(* Logix 5000 project; controller STAT 1756-L72 rev 20.12; software revision 20.04; part 23 of 34 *)
(* tags used below, declared in another part *)
   av320 : BOOL;
   BITMW2 : BOOL;
   DateTime : DINT[7];   // DINT array tag for retrieve wallclock time through GSV created during conversion
   ForceStatus : INT;   // INT tag to retrieve Force enabled value through GSV created during conversion
   FRANCK : BOOL;
   lastmonth_put1 : DINT;
   lastmonth_put2 : DINT;
   lastmonth_totosmose : DINT;
   lastmonth_totq1 : DINT;
   lastmonth_totq2 : DINT;
   lastmonth_totq3 : DINT;
   mem_vent_yesterdsay : REAL;
   memjour : DINT;
   ONS1 : DINT;
   op010 : DINT;
   passage_jourmois : BOOL;
   PM3 : BOOL;
   PM4 : BOOL;
   real : REAL;
   S_AV320_V1_FC_C : BOOL;
   S_AV320_V1_FC_O : BOOL;
   S_AV320_V2_FC_C : BOOL;
   S_AV320_V2_FC_O : BOOL;
   s_flow_lancy_L1 : REAL;
   s_flow_lancy_L2 : REAL;
   s_flow_lancy_L3 : REAL;
   s_lvl_op006 : REAL;
   s_lvl_op007 : REAL;
   s_lvl_op008 : REAL;
   s_lvl_op009 : REAL;
   s_lvl_op010 : REAL;
   s_lvl_op011 : REAL;
   s_lvl_pellets_L4 : REAL;
   s_tot_vent_day : REAL;
   scp_flow_lancy_L1 : SCP;
   scp_flow_lancy_L2 : SCP;
   scp_flow_lancy_L3 : SCP;
   scp_flvl_op006 : SCP;
   scp_flvl_op007 : SCP;
   scp_flvl_op008 : SCP;
   scp_flvl_op009 : SCP;
   scp_flvl_op010 : SCP;
   scp_flvl_op011 : SCP;
   scp_lvl_pellets_L4 : SCP;
   stat_L1 : DINT[20];
   STAT_L2 : DINT[20];
   STAT_L3 : DINT[20];
   Status : INT;   // INT tag to retrieve Status value through GSV created during conversion
   tot_pulse_venturi : REAL;
(* ibt, continued *)

ROUTINE StatusFile   (* ladder *)
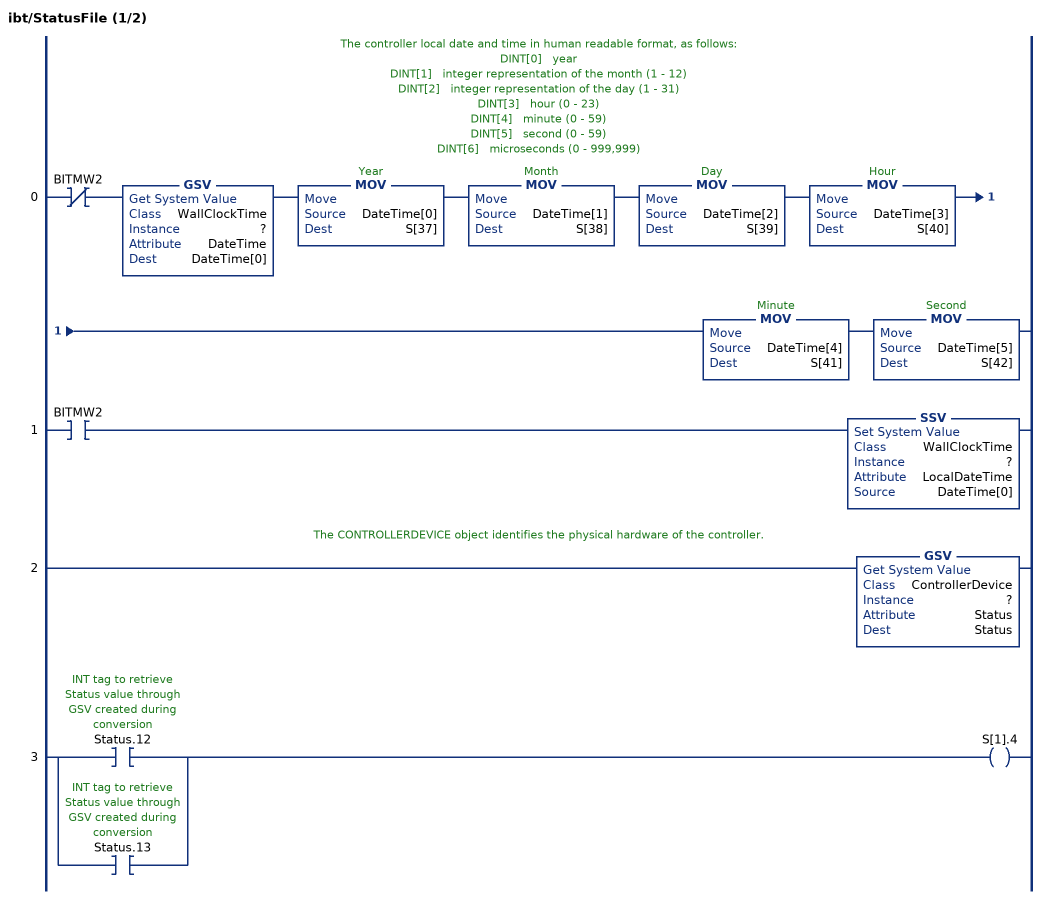
   // The controller local date and time in human readable format, as follows:
   // DINT[0] 	year
   // DINT[1] 	integer representation of the month (1 - 12)
   // DINT[2] 	integer representation of the day (1 - 31)
   // DINT[3] 	hour (0 - 23)
   // DINT[4] 	minute (0 - 59)
   // DINT[5] 	second (0 - 59)
   // DINT[6] 	microseconds (0 - 999,999)
   0: XIO(BITMW2)GSV(WallClockTime,?,DateTime,DateTime[0])MOV(DateTime[0],S[37])MOV(DateTime[1],S[38])MOV(DateTime[2],S[39])MOV(DateTime[3],S[40])MOV(DateTime[4],S[41])MOV(DateTime[5],S[42]);
   1: XIC(BITMW2)SSV(WallClockTime,?,LocalDateTime,DateTime[0]);
   // The CONTROLLERDEVICE object identifies the physical hardware of the controller.
   2: GSV(ControllerDevice,?,Status,Status);
   3: [XIC(Status.12) ,XIC(Status.13) ]OTE(S[1].4);
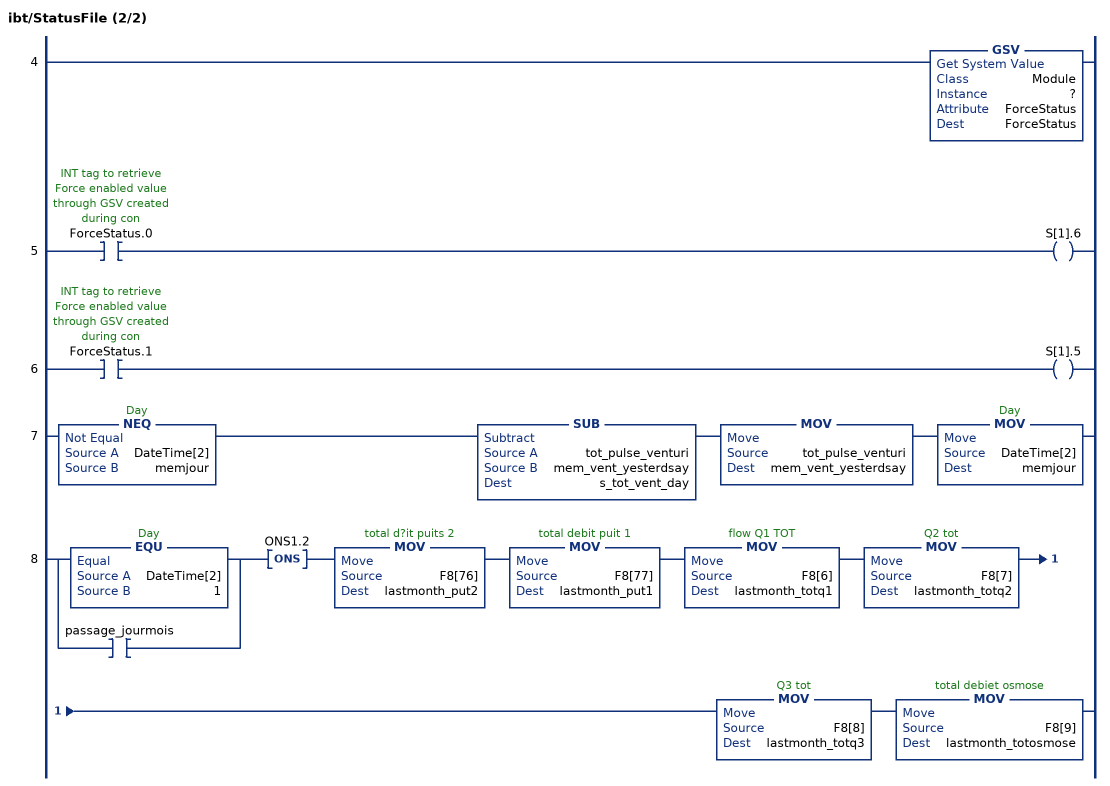
   4: GSV(Module,?,ForceStatus,ForceStatus);
   5: XIC(ForceStatus.0)OTE(S[1].6);
   6: XIC(ForceStatus.1)OTE(S[1].5);
   7: NEQ(DateTime[2],memjour)SUB(tot_pulse_venturi,mem_vent_yesterdsay,s_tot_vent_day)MOV(tot_pulse_venturi,mem_vent_yesterdsay)MOV(DateTime[2],memjour);
   8: [EQU(DateTime[2],1) ,XIC(passage_jourmois) ]ONS(ONS1.2)MOV(F8[76],lastmonth_put2)MOV(F8[77],lastmonth_put1)MOV(F8[6],lastmonth_totq1)MOV(F8[7],lastmonth_totq2)MOV(F8[8],lastmonth_totq3)MOV(F8[9],lastmonth_totosmose);
END_ROUTINE
END_PROGRAM

PROGRAM LANCY   (* main routine Lancy *)
VAR
   B3 : DINT[35] := ([1] := 2#0000_0000_0000_0000_0000_0010_0110_1001, [2] := 2#0000_0000_0000_0000_0000_0000_0000_0010, [3] := 2#0000_0000_0000_0000_0010_0001_1000_1000, [5] := 2#0000_0000_0000_0000_0000_0000_0000_0111, [6] := 2#0000_0000_0000_0000_0000_0100_0111_1110, [8] := 2#0000_0000_0000_0000_0000_0000_0000_1110, [10] := 2#0000_0000_0000_0000_1000_0000_0000_0000, [11] := 2#0000_0000_0000_0000_0000_0000_0000_1000, [25] := 2#0000_0000_0000_0000_0011_0000_0011_0000, [29] := 2#0000_0000_0000_0000_0010_0001_0000_0000, [31] := 2#0000_0000_0000_0000_0000_0100_0001_0000, [33] := 2#0000_0000_0000_0000_0000_0000_0001_1100, [34] := 2#0000_0000_0000_0000_0000_0010_0000_0000);
        [0].0   // res
        [0].1   // remplace L106E reactor tank T100 LE 106 E low level alarm
        [0].2   // remplace reactor tank T100 LE106 D
        [0].3   // remplace reactor tank T100 LE106 C
        [0].4   // remplace reactor tank T100 LE106 B
        [0].5   // remplace reactor tank T100 LE106 A
        [0].15   // ARRET POUR ENTRETIEN
        [2].0   // marche pmp puisard L123 sur debit venturi
        [2].1   // marche pmp puisard L123 sur niveau
        [2].3   // lvl orange atteint
        [2].4   // presence 1 niveau orange
        [2].5   // lvl rouge atteint
        [2].6   // changement dans les niveaux orange et rouge
        [2].7   // changement orange
        [2].8   // changement 1 niveau rouge
        [3].0   // L1 level point LE337 A
        [3].1   // L1 level point LE337 B
        [3].2   // L1 level point LE337 C
        [3].3   // L1 level point LE337 D
        [3].4   // L1 level point LE337 E
        [3].5   // L2 level point LE327 A
        [3].6   // L2 level point LE327 B
        [3].7   // L2 level point LE327 C
        [3].8   // L2 level point LE327 D
        [3].9   // L2 level point LE327 E
        [3].10   // L3 level point LE317 A
        [3].11   // L3 level point LE317 B
        [3].12   // L3 level point LE317 C
        [3].13   // L3 level point LE317 D
        [3].14   // L3 level point LE317 E
        [4].0   // L4 level point LE 400 A
        [4].1   // L4 level point LE 400 B
        [4].2   // L4 level point LE 400 C
        [4].3   // L4 level point LE 400 D
        [4].4   // L4 level point LE 400 E
        [5].0   // L4 Filtrate return Valve LV 410
        [5].1   // LV 410 open
        [5].2   // LV 410 closed
        [6].0   // op008->ph bak no default
        [6].1   // op008->holding tank no default
        [6].2   // op008->reactor no default
        [6].3   // ok L1 -> OP008
        [6].4   // ok L2 -> OP008
        [6].5   // ok L3 -> OP008
        [6].6   // ok L1->holding tank eau rinçage
        [6].7   // op008 -> L1 ok
        [6].9   // OP008 -> L3 OK
        [7].0   // pmp OP008 ok for run
        [7].3   // rinçage tuyauterie HT
        [8].0   // filtrate lift station T160 LE165 A
        [8].1   // filtrate lift station T160 LE165 B
        [8].2   // filtrate lift station T160 LE165 C
        [8].3   // filtrate lift station T160 LE165 D
        [9].0   // BP L1 -> holding tank
        [9].1   // de supervis BP L1-> OP008
        [9].2   // de superv BP L2 -> OP008
        [9].3   // de superv BP L3 -> OP008
        [9].4   // de superv BP OP008 -> reactor
        [9].6   // start].stop
        [10].11   // demande stop soude
        [10].12   // apport soude demande de marche
        [10].13   // marche soude ouverture vanne
        [10].14   // ons
        [10].15   // ons
        [25].0   // reactor tank T100 high level alarm
        [25].1   // reactor tank T100 high level alarm horn silence
        [25].2   // reactor tank T100 low level alarm
        [25].3   // reactor tank T100 low level alarm horn silence
        [25].4   // holding tank T130 low level alarm
        [25].5   // holding tank T130 low level alarm horn silence
        [25].6   // clear filtrate receiver tank T260 high level alarm
        [25].7   // clear filtrate receiver tank T260 high level alarm horn simence
        [25].10   // cloudy filtrate receiver tank T270 high level alarm
        [25].11   // cloudy filtrate receiver tank T270 high level alarm horn silence
        [25].12   // vacuum pup suction line high level alarm
        [25].13   // vacuum pup suction line high level alarm horn silence
        [25].14   // filtrate lift station high level alarm
        [25].15   // filtrate lift station high level alarm horn silence
        [26].0   // L3 high level alarm
        [26].1   // L3 high level alarm horn silence
        [26].4   // L3 low level alarm
        [26].5   // L3 low level alarm horn silence
        [26].6   // L2 high level alarm
        [26].7   // L2 high level alarm horn silence
        [26].8   // L2 low level alarm
        [26].9   // L2 low level alarm horn silence
        [26].10   // L1 high level alarm
        [26].11   // L1 high level alarm horn silence
        [26].14   // L1 low level alarm
        [26].15   // L1 low level alarm horn silence
        [27].0   // surge tank T150 turbidity control alarm
        [27].1   // surge tank T150 turbidity control alarm horn silence
        [27].2   // Mixer M110 failure alarm
        [27].3   // Mixer M110 failure alarm horn silence
        [27].4   // M120 overcurrent alarm
        [27].5   // M120 overcurrent alarm silence horn
        [27].8   // P170 overcurrent alarm
        [27].9   // P170 overcurrent alarm horn silence
        [27].10   // P180 overcurrent alarm
        [27].11   // P180 overcurrent alarm horn silence
        [27].12   // P210 overcurrent alarm
        [27].13   // P210 overcurrent alarm horn silence
        [27].14   // P220 overcurrent alarm
        [27].15   // P220 overcurrent alarm horn silence
        [28].2   // P230 overcurrent alarm
        [28].3   // P230 overcurrent alarm horn silence
        [28].4   // P240 overcurrent alarm
        [28].5   // P240 overcurrent alarm horn silence
        [28].6   // F200 overcurrent alarm
        [28].7   // F200 overcurrent alarm horn silence
        [28].8   // P250 overcurrent alarm
        [28].9   // P250 overcurrent alarm horn silence
        [28].13   // clear filtrate pumps P210 & P220 failure alarm horn silence
        [28].15   // cloudy flitrate pump P230 & P240 failure alarm horn silence
        [29].0   // filtrate lift pump P170 failure alarm
        [29].1   // filtrate lift pump P170 failure alarm horn silence
        [29].6   // 0cr
        [29].8   // 2cr
        [29].9   // 3 cr
        [29].10   // 4 cr
        [29].12   // 6 cr
        [29].13   // 7 cr
        [30].1   // 9 cr
        [30].2   // 10 CR
        [30].6   // reactor tank T100 Level B].C diffential disable relay
        [30].7   // vacuum pump P250 seal water low flow alarm
        [30].10   // vacuum pump P250 seal water low flow alarm horn silenc
        [30].11   // horn auxiliaire 1
        [30].12   // horn auxiliaire 2
        [30].13   // horn auxiliaire 3
        [30].14   // horn auxiliaire 4
        [30].15   // horn auxiliaire 5
        [31].4   // clignotant
        [31].6   // delay off timer filtrate lift pump seal water valve
        [31].7   // delay off timer filtrate lift pump P170 failure alarm
        [31].8   // tempo clear filtrate pumps seal water off delay
        [31].9   // cloudy flitrate pumps delay off timer
        [31].10   // vacuum pump P250 delay on
        [31].11   // vacuum pump seal water valve SV255 delay off timer
        [31].15   // clear filtrate pumps P210 failure alarm
        [32].0   // clear filtrate pumps P220 failure alarm
        [32].1   // tempo clear filtrate pumps P210 failure alarm delay
        [32].2   // tempo clear filtrate pumps P220 failure alarm delay
        [32].3   // cloudy flitrate pump P230 failure alarm
        [32].4   // cloudy flitrate pump P240 failure alarm
        [32].5   // cloudy flitrate pump P230 failure alarm delay
        [32].8   // cloudy flitrate pump P240 failure alarm delay
        [32].11   // vacuum pump P250 low flow delay timer
        [32].12   // shearing mixer M120 off delay timer
        [32].13   // M110 not running
        [32].14   // Mixer M110 failure delay
        [33].2   // L1 active
        [33].3   // L2 active
        [33].4   // L3 active
        [33].5   // L1 active & >level B
        [33].6   // L2 active & >level B
        [33].7   // L3 active & >level B
        [33].8   // All line not active
        [33].12   // AV valve override
        [33].13   // system high relay
        [33].14   // system high silence
        [33].15   // system high high level alarm
        [34].0   // system high high level alarm silence
        [34].1   // regenerate caustic available alarm at holding tank T130
        [34].2   // regenerate caustic available at holding tank T130 alarm silence
        [34].6   // L4 active
        [34].7   // L4 active & >level B
        [34].8   // 11 cr
        [34].9   // 12 cr
        [34].10   // L4 high level alarm
        [34].11   // L4 high level alarm horn silence
        [34].12   // L4 low level alarm
        [34].13   // L4 low level alarm horn silence
        [10].9   // demande soude station
   C5 : COUNTER[10];
        [0].DN   // g
        [0].PRE   // y
   F8 : REAL[100] := ([1] := 324.85922, [2] := 2.0, [3] := 162.42961, [4] := -2.7111664, [5] := 105.0, [10] := 199.0041, [11] := 284.0703, [12] := 333.46686, [13] := 763.174, [14] := 438.31393, [15] := 310.28265);
        [0]   // jg
        [2]   // ratio venturi].filtrat
        [3]   // debit filtrat souhaité en 0.1m³].h
        [4]   // erreur debit filtrat 0.1 m³].h
        [5]   // consigne ouverture servo vanne filtrat
        [10]   // niveau op006
        [11]   // aux niveau op007
        [12]   // aux niveau op008
        [13]   // aux niveau op009
        [14]   // aux niveau op010
        [15]   // aux niveau op011
   N20 : DINT[50] := ([0] := -16384, [1] := 4, [5] := 2, [10] := 199, [11] := 284, [12] := 333, [13] := 762, [14] := 438, [15] := 309, [17] := 632, [20] := 7935, [22] := 388, [23] := 264, [25] := 4, [30] := 5, [32] := 199, [33] := 284, [34] := 333, [35] := 199, [37] := 284, [39] := 332, [40] := -1, [41] := 766, [42] := 3, [43] := 438, [45] := 311, [46] := 1, [47] := 763, [48] := 438, [49] := 310);
        [0]   // bit pour superv
        [1]   // DEFAUT PRIORITE 1
        [2]   // defaut niveau 2
        [5].0   // DEFAULT
        [5].1   // NEW DEFAULT
        [9].1   // ack STOCK
        [10]   // niveau op006
        [11]   // niveau op007
        [12]   // niveau op008
        [13]   // niveau op009
        [14]   // niveau op010
        [15]   // niveau op011
        [16].1   // level holding tank
        [16].2   // valve positie
        [20].0   // reactor tank T100 high level alarm
        [20].1   // reactor tank T100 low level alarm
        [20].2   // holding tank T130 low level alarm
        [20].3   // clear filtrate receiver tank T260 high level alarm
        [20].4   // cloudy filtrate receiver tank T270 high level alarm
        [20].5   // vacuum pup suction line high level alarm
        [20].6   // filtrate lift station high level alarm
        [20].7   // L3 high level alarm
        [20].8   // L3 low level alarm
        [20].9   // L2 high level alarm
        [20].10   // L2 low level alarm
        [20].11   // L1 high level alarm
        [20].12   // L1 low level alarm
        [20].13   // surge tank T150 turbidity control alarm
        [20].14   // Mixer M110 failure alarm
        [20].15   // M120 overcurrent alarm
        [21].0   // P170 overcurrent alarm
        [21].1   // P180 overcurrent alarm
        [21].2   // P210 overcurrent alarm
        [21].3   // P220 overcurrent alarm
        [21].4   // P230 overcurrent alarm
        [21].5   // P240 overcurrent alarm
        [21].6   // F200 overcurrent alarm
        [21].7   // P250 overcurrent alarm
        [21].8   // filtrate lift pump P170 failure alarm
        [21].9   // vacuum pump P250 seal water low flow alarm
        [21].10   // L4 high level alarm
        [21].11   // L4 low level alarm
        [21].12   // clear filtrate pumps P210 failure alarm
        [21].13   // clear filtrate pumps P220 failure alarm
        [21].14   // cloudy flitrate pump P230 failure alarm
        [21].15   // cloudy flitrate pump P240 failure alarm
        [22].0   // system high relay
        [22].1   // system high high level alarm
        [22].2   // regenerate caustic available alarm at holding tank T130
        [22].3   // DEF POS VANNE SILO
        [22].4   // DEF POS VANNE BOUILLOIRE
        [22].5   // DEF POSIT ST VA1
        [22].6   // DEF POSIT ST VA 2
        [22].7   // DEF POSIT ST VA3
        [22].8   // DEF POSIT ST VA4
        [22].9   // DEF POSIT ST VA5
        [22].10   // DEF POSIT ST VA6
        [22].11   // DEF POSIT ST VA7
        [22].14   // DEF PP1 STAT
        [23].12   // mixer arreté pour Franck mixer stil pour herman
        [25].0   // reactor tank T100 high level alarm
        [25].1   // reactor tank T100 low level alarm
        [25].2   // holding tank T130 low level alarm
        [25].3   // clear filtrate receiver tank T260 high level alarm
        [25].4   // cloudy filtrate receiver tank T270 high level alarm
        [25].5   // vacuum pup suction line high level alarm
        [25].6   // filtrate lift station high level alarm
        [25].7   // L3 high level alarm
        [25].8   // L3 low level alarm
        [25].9   // L2 high level alarm
        [25].10   // L2 low level alarm
        [25].11   // L1 high level alarm
        [25].12   // L1 low level alarm
        [25].13   // surge tank T150 turbidity control alarm
        [25].14   // Mixer M110 failure alarm
        [25].15   // M120 overcurrent alarm
        [26].0   // P170 overcurrent alarm
        [26].1   // P180 overcurrent alarm
        [26].2   // P210 overcurrent alarm
        [26].3   // P220 overcurrent alarm
        [26].4   // P230 overcurrent alarm
        [26].5   // P240 overcurrent alarm
        [26].6   // F200 overcurrent alarm
        [26].7   // P250 overcurrent alarm
        [26].8   // filtrate lift pump P170 failure alarm
        [26].9   // vacuum pump P250 seal water low flow alarm
        [26].10   // L4 high level alarm
        [26].11   // L4 low level alarm
        [26].12   // clear filtrate pumps P210 failure alarm
        [26].13   // clear filtrate pumps P220 failure alarm
        [26].14   // cloudy flitrate pump P230 failure alarm
        [26].15   // cloudy flitrate pump P240 failure alarm
        [27].0   // system high relay
        [27].1   // system high high level alarm
        [27].2   // regenerate caustic available alarm at holding tank T130
        [27].3   // DEF POS VANNE SILO
        [27].4   // DEF POS VANNE BOUILLOIRE
        [27].5   // DEF POSIT ST VA1
        [27].6   // DEF POSIT ST VA 2
        [27].7   // DEF POSIT ST VA3
        [27].8   // DEF POSIT ST VA 4
        [27].9   // DEF POSIT ST VA5
        [27].10   // DEF POSIT ST VA6
        [27].11   // DEF POSIT ST VA7
        [27].14   // DEF PP1 STAT
        [30]   // NOMBRE DE DEFAUTS
        [31]   // MEMO NOMBRE DE DEFAUTS
        [32]   // op006
        [33]   // op007
        [34]   // op008
        [36]   // delta viveau op006
        [38]   // delta viveau op007
        [40]   // delta viveau op008
        [42]   // delta viveau op009
        [44]   // delta niveau op010
        [46]   // delta niveau op011
        [47]   // op009
        [48]   // op010
        [49]   // op011
   N7 : DINT[150] := ([1] := -250, [2] := 994, [3] := 958, [4] := -250, [5] := 982, [6] := 994, [7] := 958, [8] := 982, [10] := 165, [11] := -25, [12] := 888, [13] := 609, [15] := 955, [16] := -250, [17] := -250, [18] := 632, [19] := 269, [20] := 105, [21] := -16384, [23] := 894, [26] := 16, [29] := 525, [30] := 600, [31] := 400, [32] := 575, [33] := 350, [34] := 609, [35] := 30, [36] := 49, [37] := 65, [39] := 2, [40] := 1170, [45] := 754, [50] := 14, [57] := 10, [60] := 438, [61] := 6, [62] := 173, [64] := 20, [65] := 2048, [70] := 7, [71] := 27, [72] := 10, [73] := 11, [74] := 137, [75] := 100, [78] := 5, [90] := 6, [91] := 609, [94] := 5, [96] := 45, [98] := 45, [99] := 45, [101] := 5, [102] := 5, [103] := 5, [104] := 5, [105] := 5, [106] := 5, [110] := 8192,
        [111] := 32, [112] := 1, [113] := 7, [114] := 137, [115] := 250, [118] := 5, [140] := 21, [141] := 780, [142] := 800);
        [12]   // niveau reacteur Lancy E 905 / changer le D920 /12/07/16 C965 B975 A985
        [0]   // mojilhk
        [10]   // debit filtrat filtre-presse 0.1 m³].h
        [11]   // position servo vanne filtrat
        [13]   // niveau puisard L123
        [16]   // hac turbidity 0-1000 mtu
        [17]   // optek turbidity 0-1000 mtu
        [18]   // niveau BUFFER VOOR FILTER PERS
        [19]   // LEVEL FLITRAAT WATER FROM FILTERPERS
        [20]   // cmd position vanne filtrat
        [21]   // memo
        [25]   // vers stock quantité soude demandée
        [26].0   // vers plc stock demande de soude L1
        [26].1   // vers plc stock demande d'arret apport soude
        [26].2   // vers plc stock fc vanne apport soude décapage
        [26].3   // vers plc stock apport soude finit
        [26].4   // vers plc stock fc vanne apport soude décapage
        [29]   // niveau lift tank
        [36]   // memo debit venturi
        [38]   // diferrence debit venturi
        [45]   // soude restante
        [46].3   // de plc stock ouverture vanne soude
        [46].4   // de plc stock apport soude finit
        [46].5   // de plc stock apport soude occupé
        [46].6   // de plc stock apport soude accordé
        [46].7   // de plc stock soude vers l1
        [46].8   // de plc stock soude vers L2
        [46].9   // de plc stock soude vers L3
        [46].10   // de plc stock soude vers L4
        [46].11   // de plc stock soude vers STAT
        [50]   // debit venturi m³].h de IBT
        [51]   // reserver de IBT
        [52]   // reserver de IBT
        [53]   // reserver de IBT
        [54]   // reserver de IBT
        [55]   // reserver de IBT
        [60]   // vers ecotech op010
        [70]   // message ecriture IBT
        [90].0   // Mixer M110 failure alarm
        [90].1   // vers slc ibt marche pmp 1 puisard L123
        [90].2   // vers slc ibt marche pmp 2 puisard L123
        [90].3   // vers slc ibt stop pm3 et pm4
        [91]   // level puisard L1 2 3
        [94]   // pas à pas sequence ?? NAOH
        [95]   // DEBIT L1
        [96]   // DEBIT L2
        [97]   // DEBIT L3
        [98]   // TOTAL L 1 2 3
        [99]   // aux TOTAL L 1 2 3
        [100]   // pas à pas op008-> L4
        [101]   // pas a pas op008 -> Holding Tank
        [102]   // pas a pas op008 -> reactor
        [103]   // pas a pas L1 -> OP008
        [104]   // pas a pas L2 -> OP008
        [105]   // pas a pas L3 -> OP008
        [106]   // pas a pas renvoi eau nettoyage
        [107]   // op008 -> L1
        [108]   // op008 -> L2
        [109]   // op 008 L3
        [110]   // stock
        [131]   // MEMO AUX FLOW L1
        [132]   // MEMO AUX FLOW L2
        [133]   // MEMO AUX FLOW L2
        [134]   // MEMO AUX FLOW L3
        [135]   // MEMO AUX FLOW L3
        [140].0   // envoi defaut niv 1 present
        [140].1   // defaut niveau 2 present
        [140].2   // defaut rappel envoi
        [141]   // level high buffer fl
        [142]   // level high high buff
   N9 : DINT[200] := ([0] := 10, [1] := -1, [10] := 509, [11] := -32474, [14] := 1, [20] := 346, [21] := 1062, [23] := 4, [24] := -12, [30] := 484, [31] := 430, [33] := 4, [34] := -1, [36] := 10, [43] := 91, [60] := 2, [71] := 2349, [73] := 165, [74] := 93, [75] := -25, [76] := 609, [77] := -250, [78] := 49, [79] := 484, [80] := 199, [81] := 284, [82] := 333, [83] := 763, [84] := 438, [85] := 310, [86] := -16384, [87] := 35415, [88] := 43684, [89] := 888, [91] := 45, [94] := 930, [96] := -32346, [97] := 8614, [98] := 430, [99] := 3074, [100] := 4620, [101] := 61, [104] := 10, [107] := 270, [111] := 1, [112] := 1, [120] := 1, [121] := 1, [122] := -1, [134] := 3, [142] := 1, [143] := 9, [144] := 137, [145] := 4, [147] := 512, [148] := 5, [155] := 2, [160] := 7, [161] := 16, [162] := 1,
        [163] := 9, [164] := 137, [165] := 4, [168] := 5, [175] := 2, [180] := 7, [181] := 24, [182] := 1, [183] := 9, [184] := 137, [185] := 4, [188] := 5, [195] := 2);
        [21].0   // L2VA1 open
        [97].0   // L2VA1 open
        [100].16   // de superv Stop trajet L1 vers holding tank
        [21].1   // l2VA1 close
        [97].1   // l2VA1 close
        [97].8   // pp2 run
        [0]   // h,j;
        [0].0   // DE PLC STOCK L1 VA 4 FC O
        [0].1   // DE PLC STOCK L1 VA 4 FC F
        [0].2   // DE PLC STOCK L2 VA 4 FC O
        [0].3   // DE PLC STOCK L2 VA 4 FC F
        [2]   // de stock
        [3]   // defaut 2 stock
        [10]   // niveau decapage L1
        [11].0   // VA1 open
        [11].1   // VA1 close
        [11].2   // VA2 open
        [11].3   // VA2 close
        [11].4   // VA3 open
        [11].5   // VA3 close
        [11].6   // reserve
        [11].7   // reserve
        [11].8   // pp1 run
        [11].9   // pp1 TH
        [11].10   // pp2 run
        [11].11   // pp2 TH
        [11].12   // soude passée
        [11].14   // marche renvoi eau rinçage bain decap ligne 1
        [11].15   // arret renvoi eau rinçage bain decap ligne 1
        [12]   // total soude passé vers op008
        [14]   // reserve de ligne 1
        [20]   // level decap ligne 2
        [21].2   // L2 VA2 open
        [21].3   // VA2 close
        [21].4   // VA3 open
        [21].5   // VA3 close
        [21].6   // VA4 open
        [21].7   // VA4 close
        [21].8   // pp1 run
        [21].9   // pp1 TH
        [21].10   // pp2 run
        [21].11   // pp2 TH
        [21].12   // soude passée
        [22]   // total soude passé vers op008
        [24]   // def niv 1 L2
        [25]   // def niv 2 L2
        [30]   // niveau decapage L3
        [31].0   // VA1 open
        [31].1   // VA1 close
        [31].2   // VA2 open
        [31].3   // VA2 close
        [31].4   // VA3 open
        [31].5   // VA3 close
        [31].6   // VA4 open
        [31].7   // VA4 close
        [31].8   // pp1 run
        [31].9   // pp1 TH
        [31].10   // pp2 run
        [31].11   // pp2 TH
        [31].12   // soude passée
        [32]   // total soude passé vers op008
        [33]   // quantité eau de ligne
        [34]   // defaut niv 1 L3
        [35]   // defaut niv 2 L3
        [42]   // quantité soude demandée
        [43]   // quantite soude passé
        [50].0   // open L1VA4
        [50].1   // open L2 VA4
        [60].0   // retour alarm niv 1 vu
        [60].1   // retour alarm niv 2 vu
        [60].2   // retour alarm niv 3 vu
        [70]   // consigne en % decap L4
        [70].0   // defaut niv 1
        [71]   // conversion m³ en % dec L4
        [80]   // niveau op006
        [81]   // niveau op007
        [82]   // niveau op008
        [83]   // niveau op009
        [84]   // niveau op010
        [85]   // niveau op011
        [86].0   // lvl rouge OP006
        [86].1   // lvl orange OP006
        [86].2   // lvl rouge OP007
        [86].3   // lvl orange OP007
        [86].4   // lvl rouge OP008
        [86].5   // lvl orange OP008
        [86].6   // lvl rouge OP009
        [86].7   // lvl orange OP009
        [86].8   // lvl rouge OP010
        [86].9   // lvl orange OP010
        [86].10   // lvl rouge OP011
        [86].11   // lvl orange OP011
        [86].12   // change display spervision
        [86].13   // level op008 too low
        [87].0   // vers supervision AV 147 open
        [87].1   // vers supervision AV 320 open
        [87].2   // vers supervision LV 325 open
        [87].3   // vers supervision AV 330 open
        [87].4   // vers supervision LV 335 open
        [87].5   // vers supervision AV 310 open
        [87].6   // vers supervision LV 315 open
        [87].7   // vers supervision clear filtrate P210
        [87].8   // vers supervision clear filtrate pumps P210 failure
        [87].9   // vers supervision clear filtrate P220
        [87].10   // vers supervision clear filtrate pumpsP220 failure
        [87].11   // vers supervision cloudy filtrate P230
        [87].12   // vers supervision cloudy flitrate pump P230 failure
        [87].13   // vers supervision cloudy filtrate P240
        [87].14   // vers supervision cloudy flitrate pump P240 failure
        [87].15   // vers supervision
        [88].0   // vers supervision filtrate lift pump P170
        [88].1   // vers supervision P170 overcurrent alarm
        [88].2   // vers supervision filtrate lift pump P180
        [88].3   // vers supervision P180 overcurrent alarm
        [88].4   // vers supervision ST VA1 open
        [88].5   // vers supervision ST VA1 close
        [88].6   // vers supervision ST VA2 open
        [88].7   // vers supervision ST VA2 close
        [88].8   // vers supervision ST VA3 open
        [88].9   // vers supervision ST VA3 close
        [88].10   // vers supervision ST VA4 open
        [88].11   // vers supervision ST VA4 close
        [88].12   // vers supervision ST VA5 open
        [88].13   // vers supervision ST VA5 close
        [88].14   // vers supervision ST VA6 open
        [88].15   // vers supervision ST VA6 close
        [89]   // vers supervission niveau reacteur Lancy
        [90]   // DEBIT L1
        [91]   // DEBIT L2
        [92]   // DEBIT L3
        [93]   // level holding tank
        [94]   // level Ph bak
        [95]   // total soude passé vers op008
        [96].0   // L1 VA1 open
        [96].1   // L1 VA1 closed
        [96].2   // L1 va2 ouverte
        [96].3   // L1 va2 closed
        [96].4   // L1 va3 ouverte
        [96].5   // L1 va3 closed
        [96].6   // L1 VA4 open
        [96].7   // L1 VA4 close
        [96].8   // L1 PP1 RUN
        [97].2   // L2 VA2 open
        [97].6   // L2 VA4 open
        [97].7   // L2 VA4 close
        [98].0   // L3 VA1 open
        [98].1   // L3 VA1 closed
        [98].2   // L3 VA2 open
        [98].4   // L3 VA3 open
        [98].6   // L3 VA4 open
        [98].7   // L3 VA4 closed
        [98].8   // L3 pp1 run
        [99].0   // vers supervision ST VA7 open
        [99].1   // vers supervision ST VA7 close
        [99].2   // vers suprt defaut protection pompe PP1
        [99].3   // vers suprt rotation pompe st PP1 op008
        [99].4   // op008 - > reactor en dmd ou en rinçage
        [99].5   // op008 - > reactor run
        [99].6   // op008 - > holding tank en dmd ou en rinçage
        [99].7   // op008 - > holding tank run
        [99].8   // op008 - > phbak en demande ou en rinçage
        [99].9   // op008 - > phbak run
        [99].10   // op008 - > reactor possible
        [99].11   // op008 - > holding tank possible
        [99].12   // op008 - > phbak possible
        [99].13   // de superv BP OP008 -> reactor
        [99].14   // de superv BP op008->holding T
        [99].15   // de superv bp op008->phbak
        [100].0   // vers superv level reactor too high
        [100].1   // vers superv level holding T too high
        [100].2   // vers superv level phbak too high
        [100].3   // open].close ST VA1
        [100].4   // BP L1 -> holding tank
        [100].6   // de supervis BP L1-> OP008
        [100].7   // de superv BP L2 -> OP008
        [100].8   // de superv BP L3 -> OP008
        [101]   // stock soude pellet L4
        [102]   // res flow naoh L2
        [103]   // res flow naoh L3
        [106]   // quantité naoh demander de L3
        [110]   // total soude passé vers op008
        [111].3   // de superv bp op008 ->L1
        [111].5   // de supervision BP op008 - > L3
        [113]   // res flow naoh L1
        [123]   // memo def 1 IBT
        [124]   // stock
        [125]   // lancy
        [140]   // ligne 1
        [155].0   // open L1 VA1
        [155].1   // open L1 VA2
        [155].2   // open L1 VA3
        [155].4   // DEFAULT FLOW NaOH FROM L1
        [155].5   // DEFAULT FLOW NaOH TO L1
        [160]   // ligne2
        [175].0   // open L2 VA1
        [175].1   // open L2 VA2
        [175].2   // open L2 VA3
        [175].4   // DEFAULT FLOW NaOH FROM L2
        [175].5   // DEFAULT FLOW NaOH TO L2
        [180]   // ligne 3
        [195].0   // open L3 VA1
        [195].1   // open L3 VA2
        [195].2   // open L3 VA3
        [195].3   // open L3 VA4
        [195].4   // DEFAULT FLOW NaOH FROM L3
        [195].5   // DEFAULT FLOW NaOH TO L3
        [195].6   // reactor tank T100 HH vers L3
   R6 : CONTROL[10];
   S : INT[164] := ([0] := 16#0004, [1] := 16#00e6, [2] := 16#9012, [3] := 16#a001, [4] := 16#4c06, [5] := 16#4000, [6] := 16#0021, [11] := 16#ffff, [12] := 16#ffff, [14] := 16#0046, [15] := 16#0b1e, [17] := 16#0002, [21] := 16#0002, [22] := 16#0003, [23] := 16#0001, [27] := 16#ffff, [28] := 16#ffff, [33] := 16#1808, [34] := 16#0002, [35] := 16#000b, [37] := 16#0775, [38] := 16#000c, [39] := 16#0018, [40] := 16#0006, [41] := 16#0021, [42] := 16#0008, [53] := 16#0006, [54] := 16#0021, [57] := 16#0191, [58] := 16#0002, [59] := 16#0006, [60] := 16#021d, [61] := 16#0002, [62] := 16#0007, [63] := 16#0401, [64] := 16#005f, [65] := 16#0010, [66] := 16#0200, [83] := 16#0046, [84] := 16#f000, [85] := 16#0001, [86] := 16#01a3);
   T4 : TIMER[100] := ([0].PRE := 9999, [0].ACC := 45, [1].PRE := 5000, [2].PRE := 10000, [3].PRE := 5000, [4].PRE := 5000, [5].PRE := 5000, [6].PRE := 5000, [7].PRE := 5000, [8].PRE := 5000, [9].PRE := 3000, [9].ACC := 3000, [9].EN := 1, [9].DN := 1, [10].PRE := 5000, [11].PRE := 3000, [12].PRE := 60000, [12].ACC := 50750, [12].EN := 1, [12].TT := 1, [13].PRE := 5000, [14].PRE := 2000, [14].ACC := 1500, [14].EN := 1, [14].TT := 1, [15].PRE := 10000, [15].ACC := 4000, [15].EN := 1, [15].TT := 1, [16].PRE := 60000, [16].ACC := 60000, [17].PRE := 450000, [18].PRE := 1200000, [18].ACC := 936100, [18].TT := 1, [18].DN := 1, [19].PRE := 30000, [19].ACC := 23850, [19].EN := 1, [19].TT := 1, [20].PRE := 700, [20].ACC := 600, [20].EN := 1, [20].TT := 1, [21].PRE := 5000, [22].PRE := 50000, [23].PRE := 50000, [24].PRE := 10000, [25].PRE := 5000, [26].PRE := 90000, [27].PRE := 3000, [27].ACC := 600, [27].EN := 1, [27].TT := 1, [28].PRE := 150000, [29].PRE := 150000, [30].PRE := 120000, [31].PRE := 5000, [32].PRE := 150000, [33].PRE := 150000,
        [34].PRE := 150000, [35].PRE := 20000, [35].ACC := 20000, [35].EN := 1, [35].DN := 1, [36].PRE := 20000, [36].ACC := 20000, [36].EN := 1, [36].DN := 1, [37].PRE := 30000, [38].PRE := 240000, [39].PRE := 240000, [40].PRE := 240000, [41].PRE := 240000, [42].PRE := 240000, [43].PRE := 240000, [44].PRE := 5000, [45].PRE := 60000, [46].PRE := 60000, [47].PRE := 60000, [48].PRE := 120000, [49].PRE := 60000, [50].PRE := 60000, [51].PRE := 60000, [52].PRE := 60000, [53].PRE := 60000, [54].PRE := 60000, [54].ACC := 50650, [54].EN := 1, [54].TT := 1, [55].PRE := 60000, [56].PRE := 60000, [57].PRE := 60000, [58].PRE := 5000, [58].ACC := 5000, [59].PRE := 1200000, [59].ACC := 1200000, [59].EN := 1, [59].DN := 1, [60].PRE := 300000, [61].PRE := 600000, [62].PRE := 30000, [63].PRE := 30000, [64].PRE := 300000, [64].ACC := 300000, [65].PRE := 2000, [65].EN := 1, [65].DN := 1, [66].PRE := 2000, [66].ACC := 2000, [68].PRE := 3000, [68].ACC := 3000, [69].PRE := 3000, [69].EN := 1, [69].DN := 1, [70].PRE := 31000000, [70].ACC := 399000, [71].PRE := 2000, [71].EN := 1, [71].DN := 1,
        [72].PRE := 2000);
        [0]   // kghkh;
        [1]   // delay off timer filtrate lift pump seal water valve SV 175
        [1].DN   // timer filtrate lift pump seal water valve SV 175
        [2]   // delay off timer filtrate lift pump P170 failure alarm
        [3]   // clear filtrate pumps seal water off delay
        [4]   // clear filtrate pumps P210 failure alarm delay
        [5]   // clear filtrate pumps P220 failure alarm delay
        [6]   // timer cloudy flitrate pumps delay off
        [7]   // timer cloudy flitrate pump P230 failure alarm delay
        [8]   // timer cloudy flitrate pump P240 failure alarm delay
        [9]   // timer vacuum pump P250 delay on
        [10]   // timer vacuum pump seal water valve SV255 delay off
        [11]   // timer vacuum pump P250 low flow delay
        [12]   // timer shearing mixer M120 off delay
        [13]   // timer Mixer M110 failure delay
        [14]   // tempo clignotant
        [15]   // tempo envoi message to ibt
        [16]   // remplissage eau T100 apres level D
        [17]   // temps mini marche pmp puisard L123
        [18]   // temps entre 2 marche pmp puisard L123
        [19]   // tempo sample debit venturi
        [20]   // fréquence update consigne servo vanne filtrat
        [21]   // tempo stop pompe STPP1
        [22]   // rinse delay
        [27]   // TEMPO MSG
        [28]   // temps rinçage tuyauterie depuis L1
        [29]   // temps rinçage tuyauterie depuis L2
        [30]   // temps rinçage tuyauterie depuis L3
        [34]   // tempo rinçage op008->L3
        [39]   // FLOW L1 DISAPEARED
        [40]   // FLOW L2 DISAPEARED
        [41]   // FLOW L2 DISAPEARED
        [42]   // FLOW L3 DISAPEARED
        [43]   // FLOW L3 DISAPEARED
        [44]   // redemarrage ST VA2
        [45]   // DEF POS VANNE SILO
        [46]   // DEF POS VANNE BOUILLOIRE
        [47]   // DEF POSIT ST VA1
        [48]   // DEF POSIT ST VA 2
        [49]   // DEF POSIT ST VA3
        [50]   // DEF POSIT ST VA4
        [51]   // DEF POSIT ST VA5
        [52]   // DEF POSIT ST VA6
        [53]   // DEF POSIT ST VA7
        [54]   // tempo 1 min
        [55]   // envoi 1 min boue au
        [58]   // redemarrage ST VA2
        [59]   // tempo low low level pisard L1 2 3
        [61]   // base temps mouvement vanne pour eviter blocage
        [62]   // tempo mouvement vanne pour eviter blocage
        [64]   // trajet refusé
END_VAR

ROUTINE Lancy   (* ladder *)
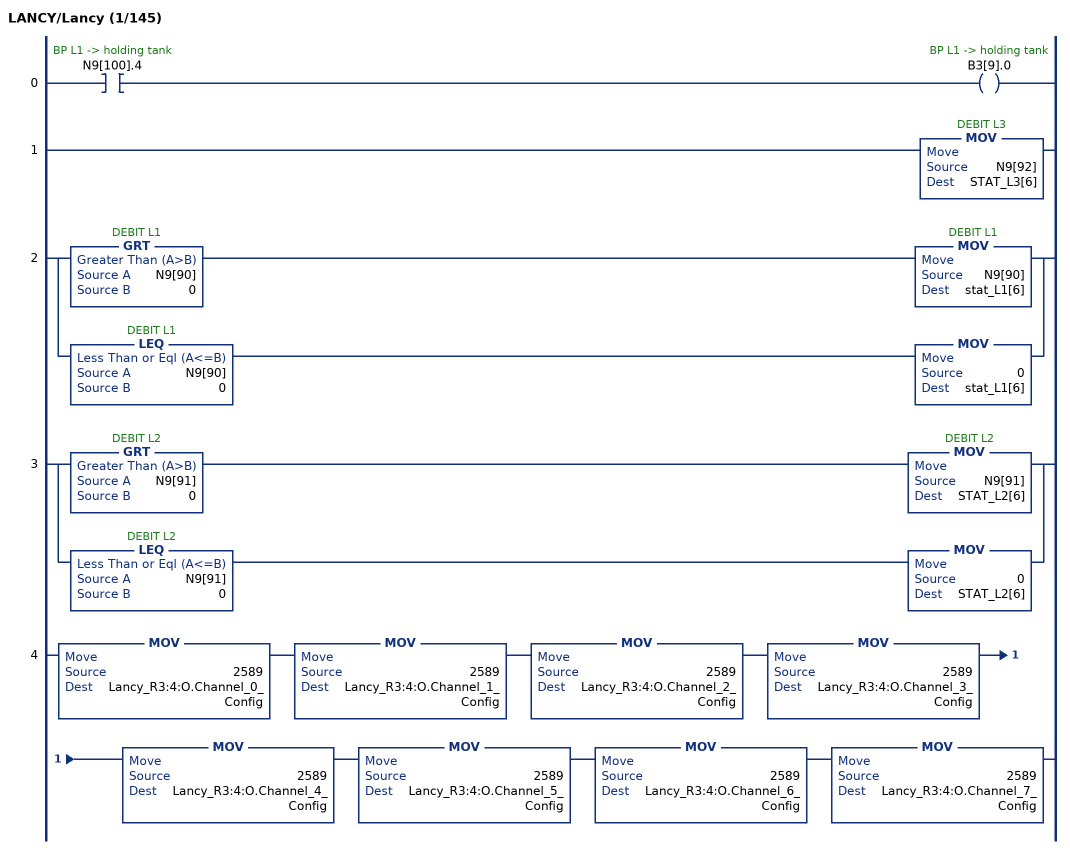
   0: XIC(N9[100].4)OTE(B3[9].0);
   1: MOV(N9[92],STAT_L3[6]);
   2: [GRT(N9[90],0) MOV(N9[90],stat_L1[6]) ,LEQ(N9[90],0) MOV(0,stat_L1[6]) ];
   3: [GRT(N9[91],0) MOV(N9[91],STAT_L2[6]) ,LEQ(N9[91],0) MOV(0,STAT_L2[6]) ];
   4: MOV(2589,Lancy_R3:4:O.Channel_0_Config)MOV(2589,Lancy_R3:4:O.Channel_1_Config)MOV(2589,Lancy_R3:4:O.Channel_2_Config)MOV(2589,Lancy_R3:4:O.Channel_3_Config)MOV(2589,Lancy_R3:4:O.Channel_4_Config)MOV(2589,Lancy_R3:4:O.Channel_5_Config)MOV(2589,Lancy_R3:4:O.Channel_6_Config)MOV(2589,Lancy_R3:4:O.Channel_7_Config);
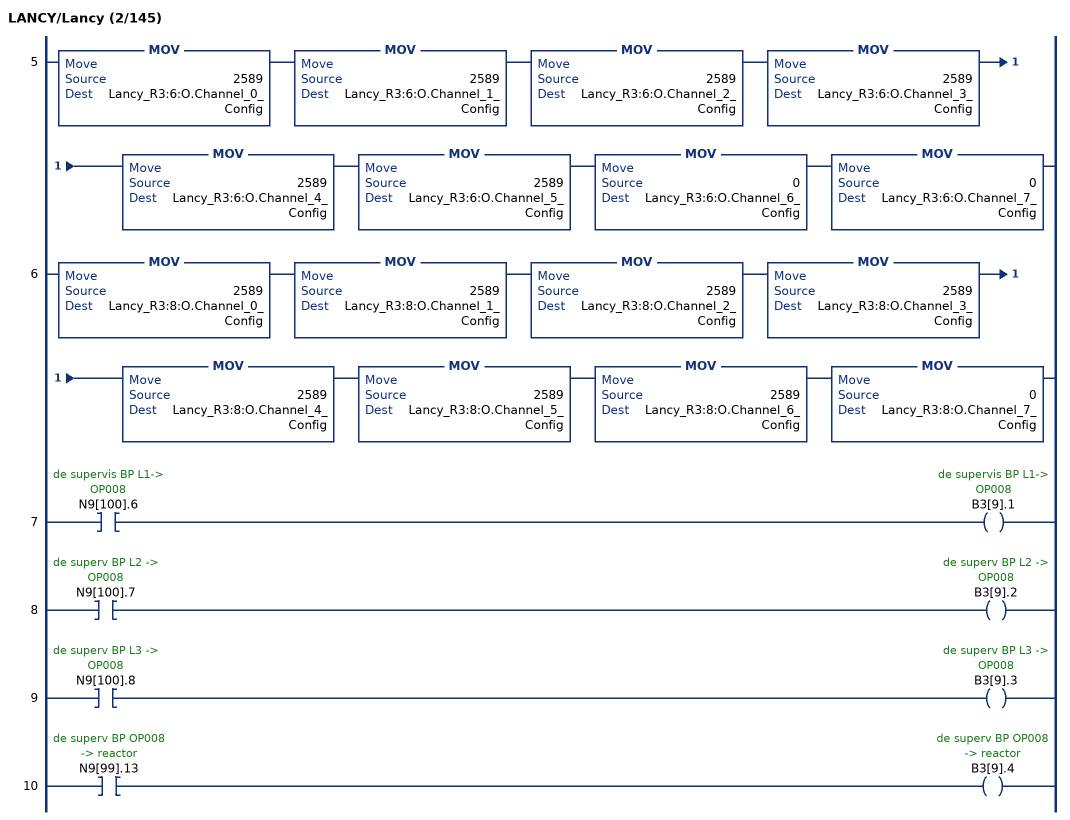
   5: MOV(2589,Lancy_R3:6:O.Channel_0_Config)MOV(2589,Lancy_R3:6:O.Channel_1_Config)MOV(2589,Lancy_R3:6:O.Channel_2_Config)MOV(2589,Lancy_R3:6:O.Channel_3_Config)MOV(2589,Lancy_R3:6:O.Channel_4_Config)MOV(2589,Lancy_R3:6:O.Channel_5_Config)MOV(0,Lancy_R3:6:O.Channel_6_Config)MOV(0,Lancy_R3:6:O.Channel_7_Config);
   6: MOV(2589,Lancy_R3:8:O.Channel_0_Config)MOV(2589,Lancy_R3:8:O.Channel_1_Config)MOV(2589,Lancy_R3:8:O.Channel_2_Config)MOV(2589,Lancy_R3:8:O.Channel_3_Config)MOV(2589,Lancy_R3:8:O.Channel_4_Config)MOV(2589,Lancy_R3:8:O.Channel_5_Config)MOV(2589,Lancy_R3:8:O.Channel_6_Config)MOV(0,Lancy_R3:8:O.Channel_7_Config);
   7: XIC(N9[100].6)OTE(B3[9].1);
   8: XIC(N9[100].7)OTE(B3[9].2);
   9: XIC(N9[100].8)OTE(B3[9].3);
   10: XIC(N9[99].13)OTE(B3[9].4);
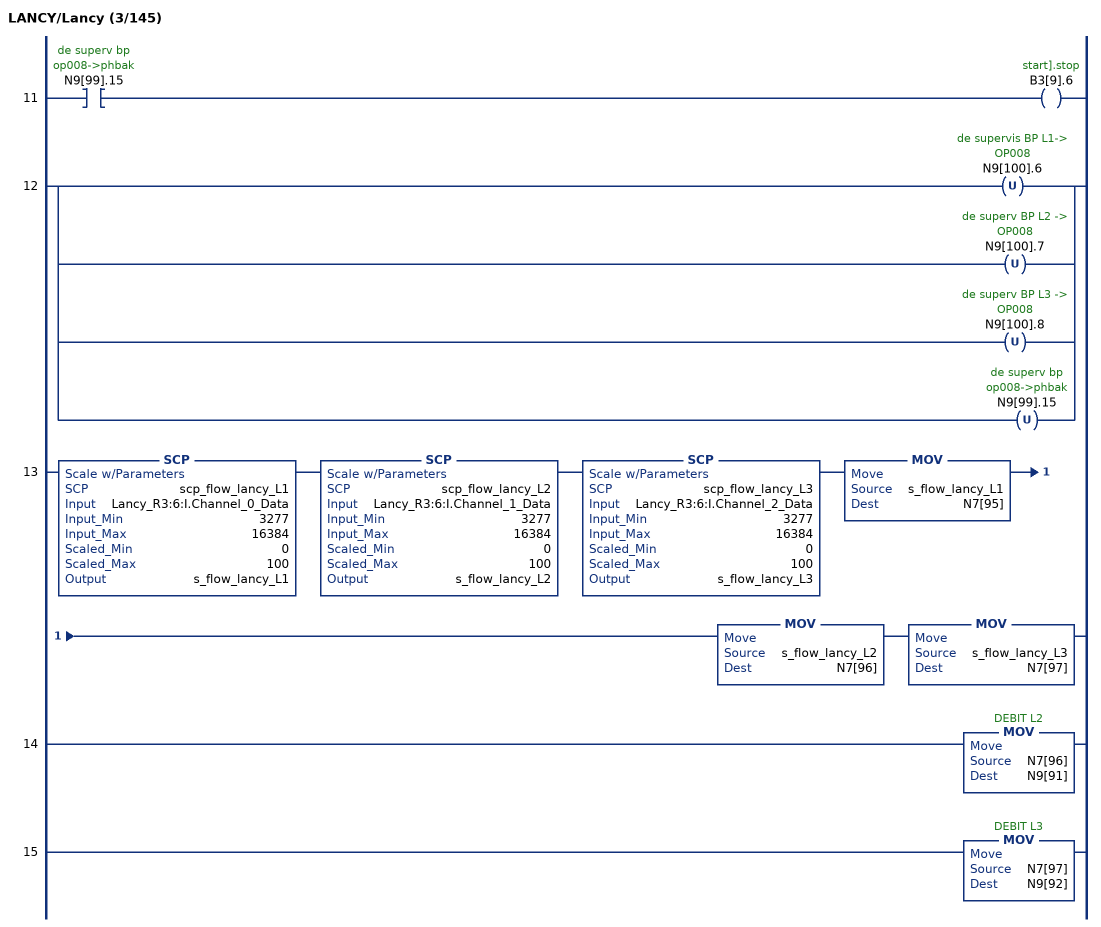
   11: XIC(N9[99].15)OTE(B3[9].6);
   12: [OTU(N9[100].6) ,OTU(N9[100].7) ,OTU(N9[100].8) ,OTU(N9[99].15) ];
   13: SCP(scp_flow_lancy_L1,Lancy_R3:6:I.Channel_0_Data,3277,16384,0,100,s_flow_lancy_L1)SCP(scp_flow_lancy_L2,Lancy_R3:6:I.Channel_1_Data,3277,16384,0,100,s_flow_lancy_L2)SCP(scp_flow_lancy_L3,Lancy_R3:6:I.Channel_2_Data,3277,16384,0,100,s_flow_lancy_L3)MOV(s_flow_lancy_L1,N7[95])MOV(s_flow_lancy_L2,N7[96])MOV(s_flow_lancy_L3,N7[97]);
   14: MOV(N7[96],N9[91]);
   15: MOV(N7[97],N9[92]);
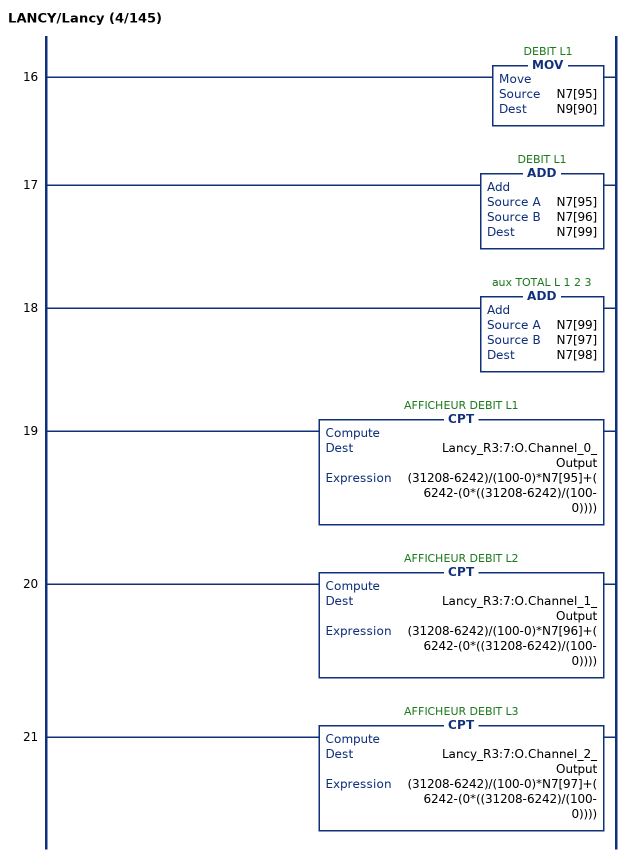
   16: MOV(N7[95],N9[90]);
   17: ADD(N7[95],N7[96],N7[99]);
   18: ADD(N7[99],N7[97],N7[98]);
   19: CPT(Lancy_R3:7:O.Channel_0_Output,(31208-6242)/(100-0)*N7[95]+(6242-(0*((31208-6242)/(100-0)))));
   20: CPT(Lancy_R3:7:O.Channel_1_Output,(31208-6242)/(100-0)*N7[96]+(6242-(0*((31208-6242)/(100-0)))));
   21: CPT(Lancy_R3:7:O.Channel_2_Output,(31208-6242)/(100-0)*N7[97]+(6242-(0*((31208-6242)/(100-0)))));
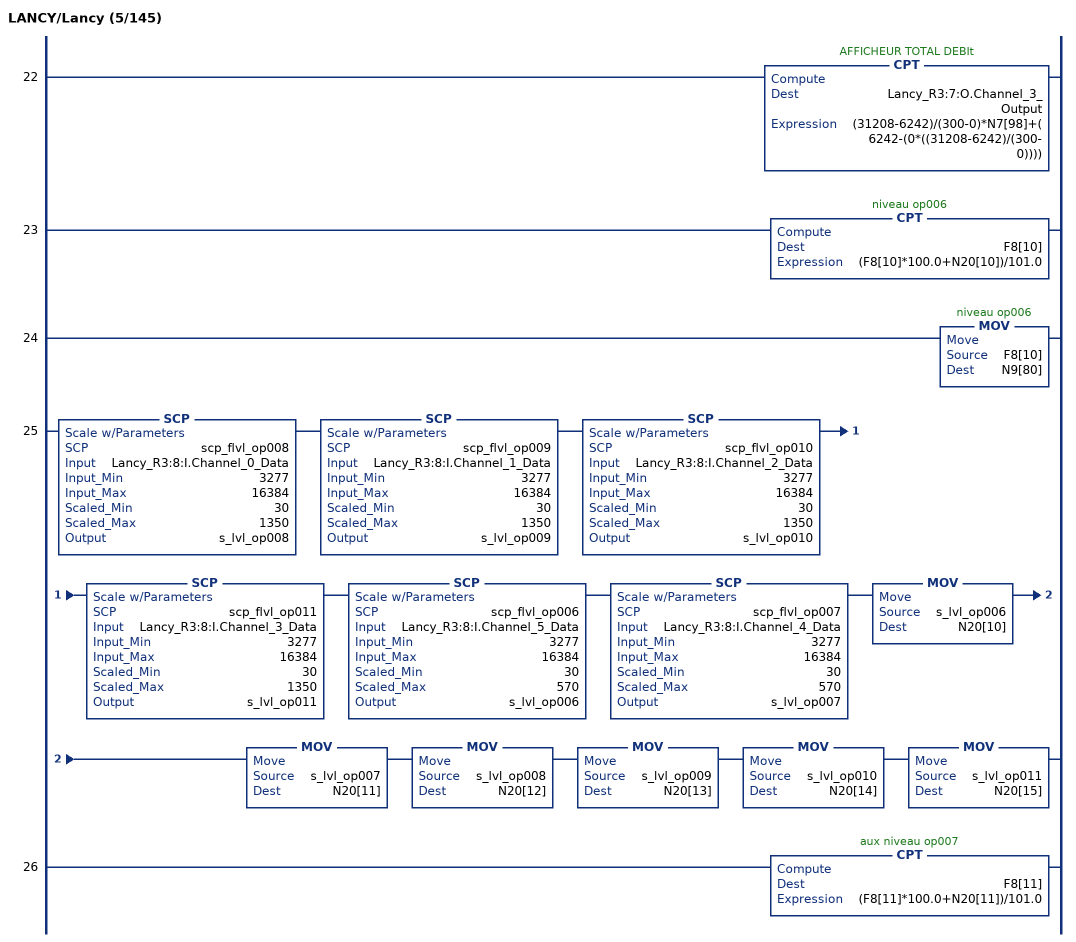
   22: CPT(Lancy_R3:7:O.Channel_3_Output,(31208-6242)/(300-0)*N7[98]+(6242-(0*((31208-6242)/(300-0)))));
   23: CPT(F8[10],(F8[10]*100.0+N20[10])/101.0);
   24: MOV(F8[10],N9[80]);
   25: SCP(scp_flvl_op008,Lancy_R3:8:I.Channel_0_Data,3277,16384,30,1350,s_lvl_op008)SCP(scp_flvl_op009,Lancy_R3:8:I.Channel_1_Data,3277,16384,30,1350,s_lvl_op009)SCP(scp_flvl_op010,Lancy_R3:8:I.Channel_2_Data,3277,16384,30,1350,s_lvl_op010)SCP(scp_flvl_op011,Lancy_R3:8:I.Channel_3_Data,3277,16384,30,1350,s_lvl_op011)SCP(scp_flvl_op006,Lancy_R3:8:I.Channel_5_Data,3277,16384,30,570,s_lvl_op006)SCP(scp_flvl_op007,Lancy_R3:8:I.Channel_4_Data,3277,16384,30,570,s_lvl_op007)MOV(s_lvl_op006,N20[10])MOV(s_lvl_op007,N20[11])MOV(s_lvl_op008,N20[12])MOV(s_lvl_op009,N20[13])MOV(s_lvl_op010,N20[14])MOV(s_lvl_op011,N20[15]);
   26: CPT(F8[11],(F8[11]*100.0+N20[11])/101.0);
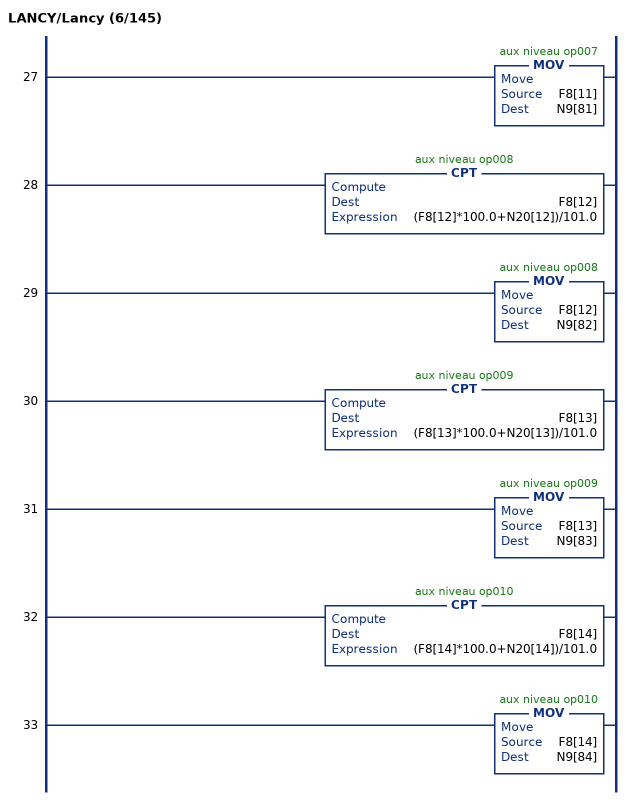
   27: MOV(F8[11],N9[81]);
   28: CPT(F8[12],(F8[12]*100.0+N20[12])/101.0);
   29: MOV(F8[12],N9[82]);
   30: CPT(F8[13],(F8[13]*100.0+N20[13])/101.0);
   31: MOV(F8[13],N9[83]);
   32: CPT(F8[14],(F8[14]*100.0+N20[14])/101.0);
   33: MOV(F8[14],N9[84]);
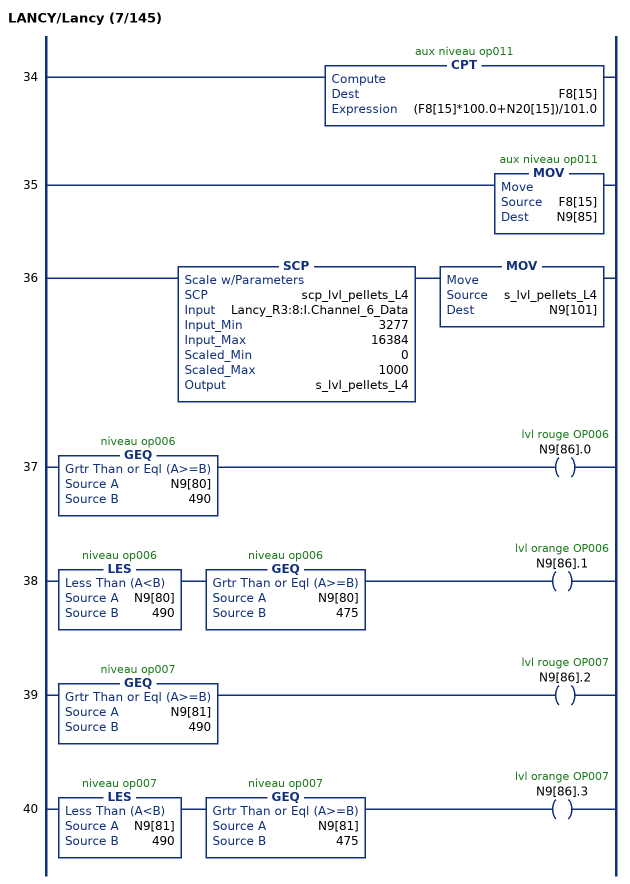
   34: CPT(F8[15],(F8[15]*100.0+N20[15])/101.0);
   35: MOV(F8[15],N9[85]);
   36: SCP(scp_lvl_pellets_L4,Lancy_R3:8:I.Channel_6_Data,3277,16384,0,1000,s_lvl_pellets_L4)MOV(s_lvl_pellets_L4,N9[101]);
   37: GEQ(N9[80],490)OTE(N9[86].0);
   38: LES(N9[80],490)GEQ(N9[80],475)OTE(N9[86].1);
   39: GEQ(N9[81],490)OTE(N9[86].2);
   40: LES(N9[81],490)GEQ(N9[81],475)OTE(N9[86].3);
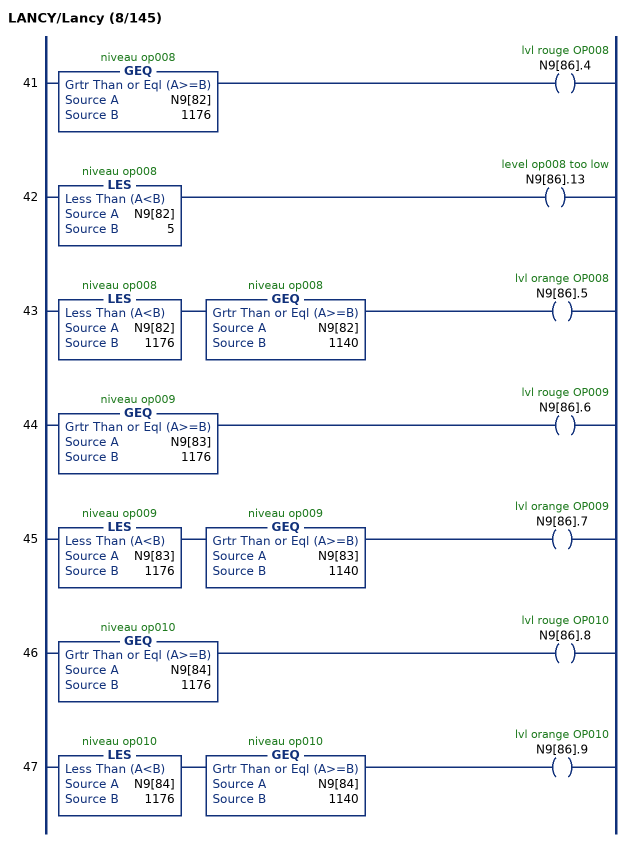
   41: GEQ(N9[82],1176)OTE(N9[86].4);
   42: LES(N9[82],5)OTE(N9[86].13);
   43: LES(N9[82],1176)GEQ(N9[82],1140)OTE(N9[86].5);
   44: GEQ(N9[83],1176)OTE(N9[86].6);
   45: LES(N9[83],1176)GEQ(N9[83],1140)OTE(N9[86].7);
   46: GEQ(N9[84],1176)OTE(N9[86].8);
   47: LES(N9[84],1176)GEQ(N9[84],1140)OTE(N9[86].9);
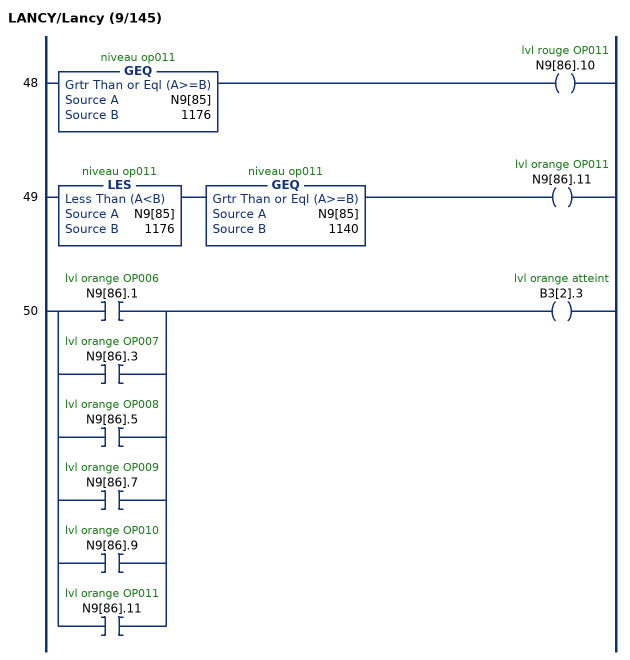
   48: GEQ(N9[85],1176)OTE(N9[86].10);
   49: LES(N9[85],1176)GEQ(N9[85],1140)OTE(N9[86].11);
   50: [XIC(N9[86].1) ,XIC(N9[86].3) ,XIC(N9[86].5) ,XIC(N9[86].7) ,XIC(N9[86].9) ,XIC(N9[86].11) ]OTE(B3[2].3);
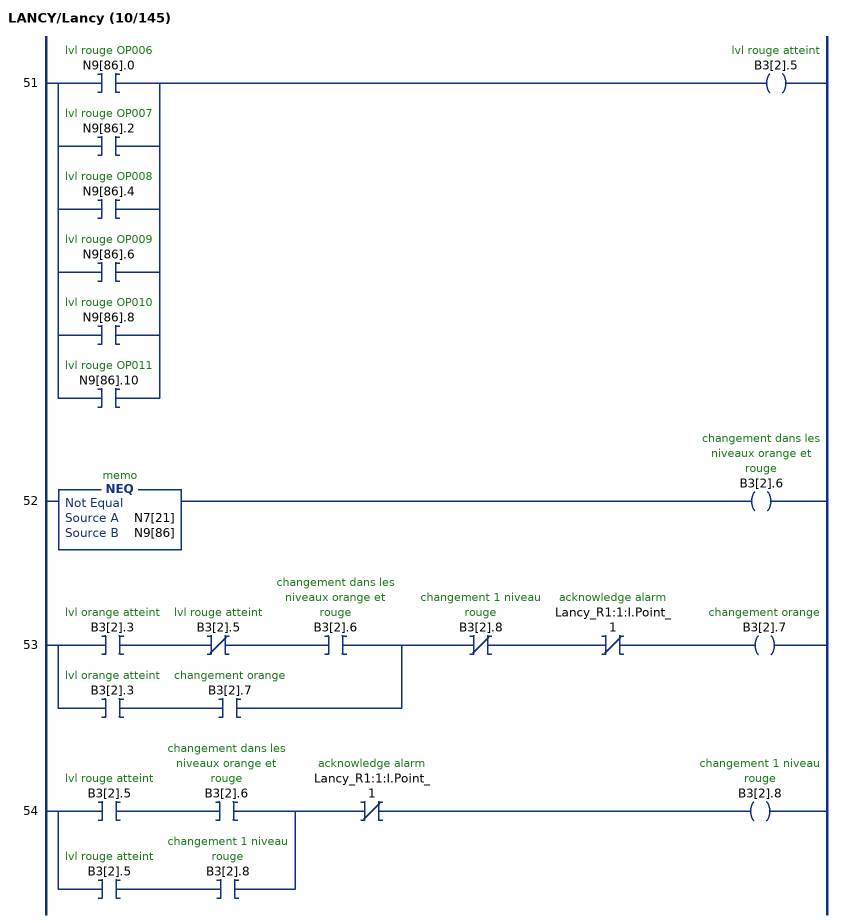
   51: [XIC(N9[86].0) ,XIC(N9[86].2) ,XIC(N9[86].4) ,XIC(N9[86].6) ,XIC(N9[86].8) ,XIC(N9[86].10) ]OTE(B3[2].5);
   52: NEQ(N7[21],N9[86])OTE(B3[2].6);
   53: [XIC(B3[2].3) XIO(B3[2].5) XIC(B3[2].6) ,XIC(B3[2].3) XIC(B3[2].7) ]XIO(B3[2].8)XIO(Lancy_R1:1:I.Point_1)OTE(B3[2].7);
   54: [XIC(B3[2].5) XIC(B3[2].6) ,XIC(B3[2].5) XIC(B3[2].8) ]XIO(Lancy_R1:1:I.Point_1)OTE(B3[2].8);
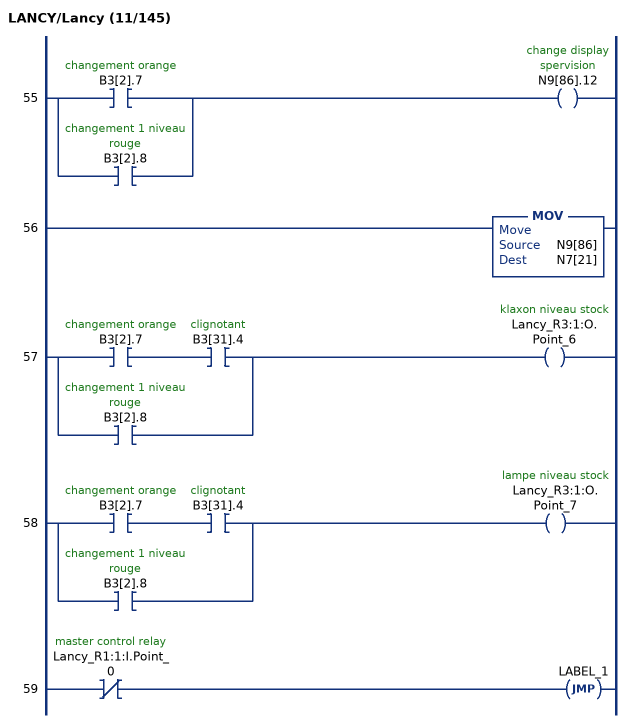
   55: [XIC(B3[2].7) ,XIC(B3[2].8) ]OTE(N9[86].12);
   56: MOV(N9[86],N7[21]);
   57: [XIC(B3[2].7) XIC(B3[31].4) ,XIC(B3[2].8) ]OTE(Lancy_R3:1:O.Point_6);
   58: [XIC(B3[2].7) XIC(B3[31].4) ,XIC(B3[2].8) ]OTE(Lancy_R3:1:O.Point_7);
   59: XIO(Lancy_R1:1:I.Point_0)JMP(LABEL_1);
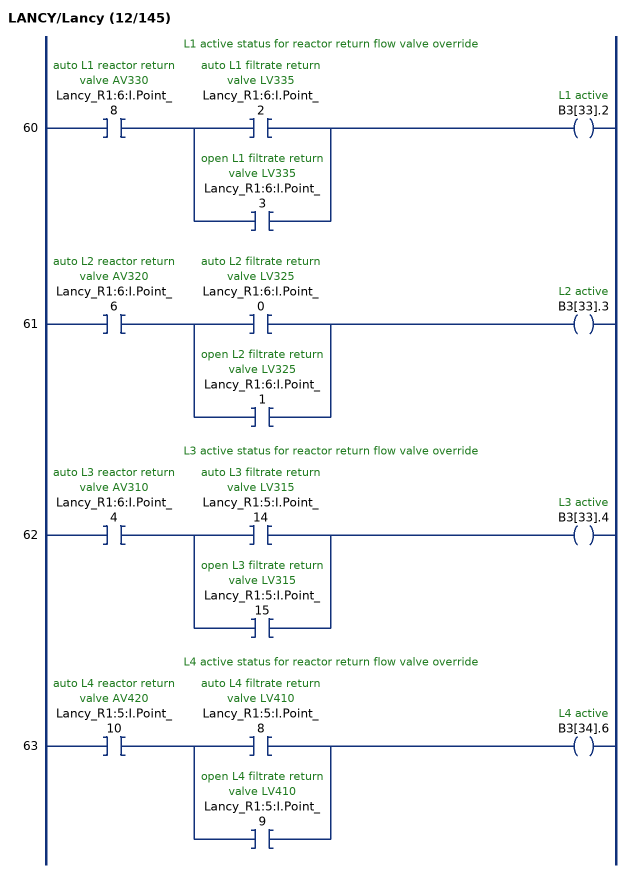
   // L1 active status for reactor return flow valve override
   60: XIC(Lancy_R1:6:I.Point_8)[XIC(Lancy_R1:6:I.Point_2) ,XIC(Lancy_R1:6:I.Point_3) ]OTE(B3[33].2);
   61: XIC(Lancy_R1:6:I.Point_6)[XIC(Lancy_R1:6:I.Point_0) ,XIC(Lancy_R1:6:I.Point_1) ]OTE(B3[33].3);
   // L3 active status for reactor return flow valve override
   62: XIC(Lancy_R1:6:I.Point_4)[XIC(Lancy_R1:5:I.Point_14) ,XIC(Lancy_R1:5:I.Point_15) ]OTE(B3[33].4);
   // L4 active status for reactor return flow valve override
   63: XIC(Lancy_R1:5:I.Point_10)[XIC(Lancy_R1:5:I.Point_8) ,XIC(Lancy_R1:5:I.Point_9) ]OTE(B3[34].6);
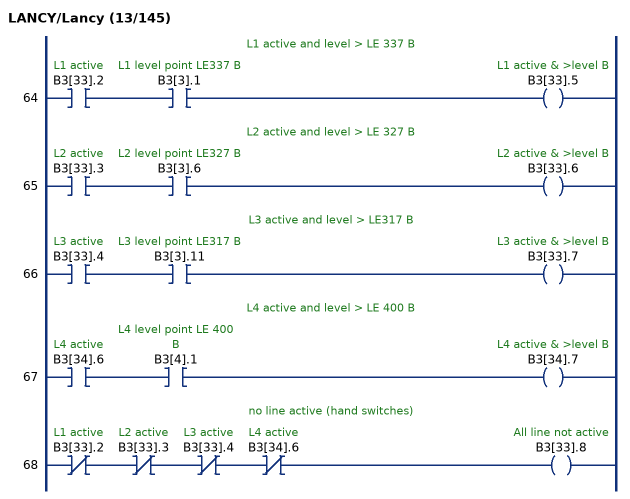
   // L1 active and level > LE 337 B
   64: XIC(B3[33].2)XIC(B3[3].1)OTE(B3[33].5);
   // L2 active and level > LE 327 B
   65: XIC(B3[33].3)XIC(B3[3].6)OTE(B3[33].6);
   // L3 active and level > LE317 B
   66: XIC(B3[33].4)XIC(B3[3].11)OTE(B3[33].7);
   // L4 active and level > LE 400 B
   67: XIC(B3[34].6)XIC(B3[4].1)OTE(B3[34].7);
   // no line active (hand switches)
   68: XIO(B3[33].2)XIO(B3[33].3)XIO(B3[33].4)XIO(B3[34].6)OTE(B3[33].8);
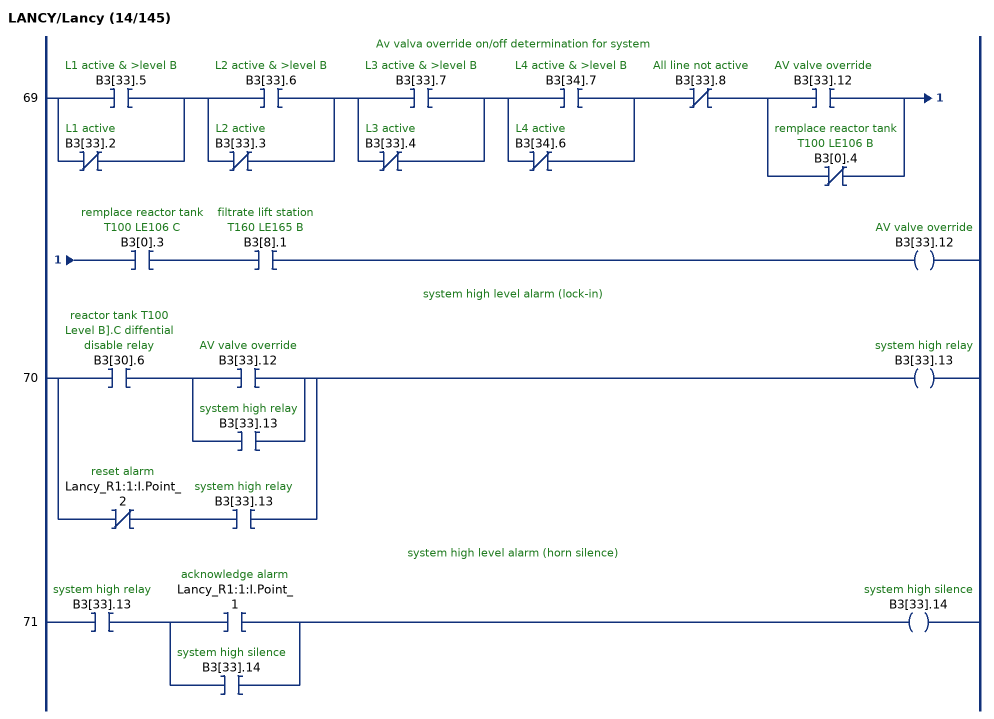
   // Av valva override on/off determination for system
   69: [XIC(B3[33].5) ,XIO(B3[33].2) ][XIC(B3[33].6) ,XIO(B3[33].3) ][XIC(B3[33].7) ,XIO(B3[33].4) ][XIC(B3[34].7) ,XIO(B3[34].6) ]XIO(B3[33].8)[XIC(B3[33].12) ,XIO(B3[0].4) ]XIC(B3[0].3)XIC(B3[8].1)OTE(B3[33].12);
   // system high level alarm (lock-in)
   70: [XIC(B3[30].6) [XIC(B3[33].12) ,XIC(B3[33].13) ] ,XIO(Lancy_R1:1:I.Point_2) XIC(B3[33].13) ]OTE(B3[33].13);
   // system high level alarm (horn silence)
   71: XIC(B3[33].13)[XIC(Lancy_R1:1:I.Point_1) ,XIC(B3[33].14) ]OTE(B3[33].14);
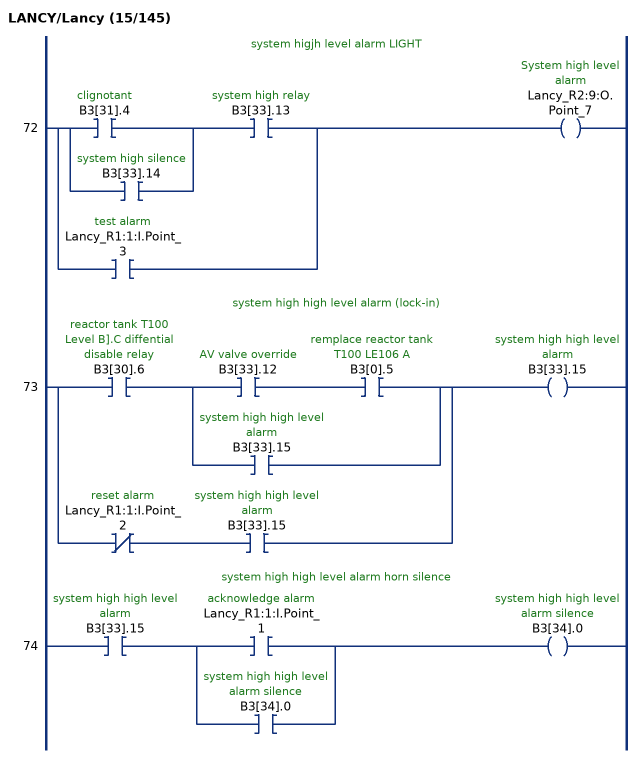
   // system higjh level alarm LIGHT
   72: [[XIC(B3[31].4) ,XIC(B3[33].14) ] XIC(B3[33].13) ,XIC(Lancy_R1:1:I.Point_3) ]OTE(Lancy_R2:9:O.Point_7);
   // system high high level alarm (lock-in)
   73: [XIC(B3[30].6) [XIC(B3[33].12) XIC(B3[0].5) ,XIC(B3[33].15) ] ,XIO(Lancy_R1:1:I.Point_2) XIC(B3[33].15) ]OTE(B3[33].15);
   // system high high level alarm horn silence
   74: XIC(B3[33].15)[XIC(Lancy_R1:1:I.Point_1) ,XIC(B3[34].0) ]OTE(B3[34].0);
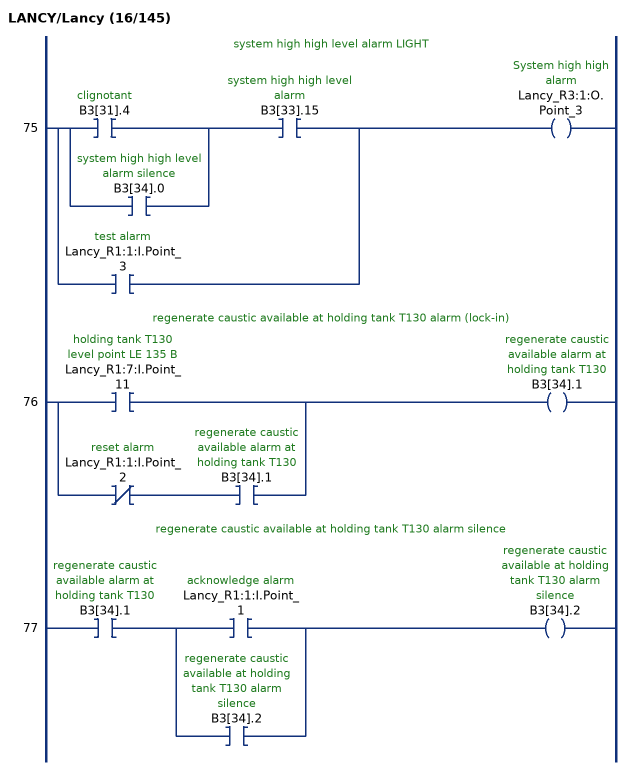
   // system high high level alarm LIGHT
   75: [[XIC(B3[31].4) ,XIC(B3[34].0) ] XIC(B3[33].15) ,XIC(Lancy_R1:1:I.Point_3) ]OTE(Lancy_R3:1:O.Point_3);
   // regenerate caustic available at holding tank T130 alarm (lock-in)
   76: [XIC(Lancy_R1:7:I.Point_11) ,XIO(Lancy_R1:1:I.Point_2) XIC(B3[34].1) ]OTE(B3[34].1);
   // regenerate caustic available at holding tank T130 alarm silence
   77: XIC(B3[34].1)[XIC(Lancy_R1:1:I.Point_1) ,XIC(B3[34].2) ]OTE(B3[34].2);
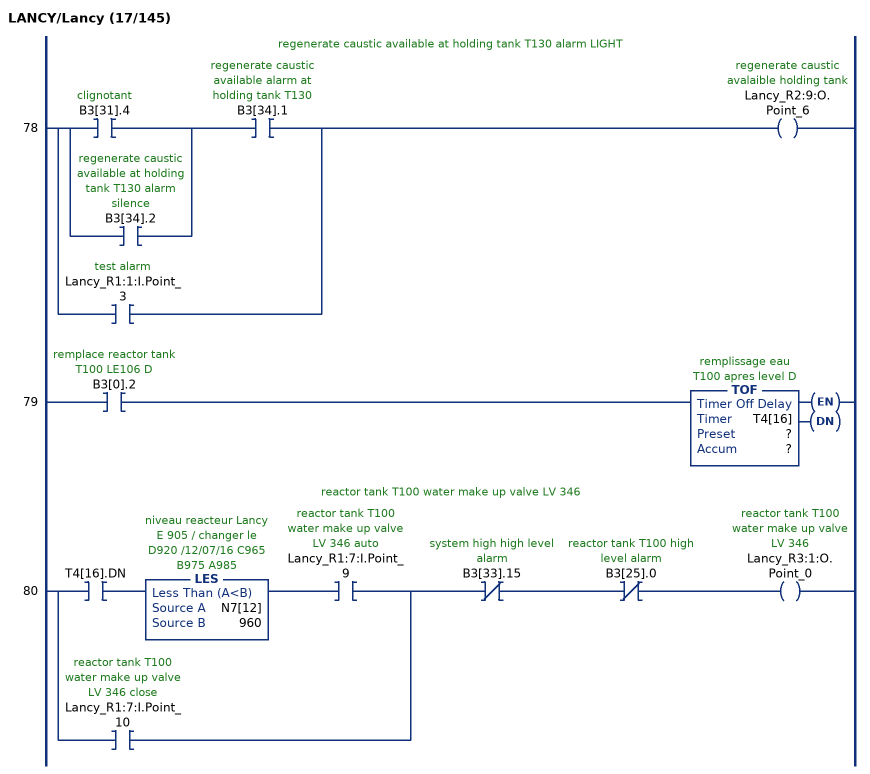
   // regenerate caustic available at holding tank T130 alarm LIGHT
   78: [[XIC(B3[31].4) ,XIC(B3[34].2) ] XIC(B3[34].1) ,XIC(Lancy_R1:1:I.Point_3) ]OTE(Lancy_R2:9:O.Point_6);
   79: XIC(B3[0].2)TOF(T4[16],?,?);
   // reactor tank T100 water make up valve LV 346
   80: [XIC(T4[16].DN) LES(N7[12],960) XIC(Lancy_R1:7:I.Point_9) ,XIC(Lancy_R1:7:I.Point_10) ]XIO(B3[33].15)XIO(B3[25].0)OTE(Lancy_R3:1:O.Point_0);
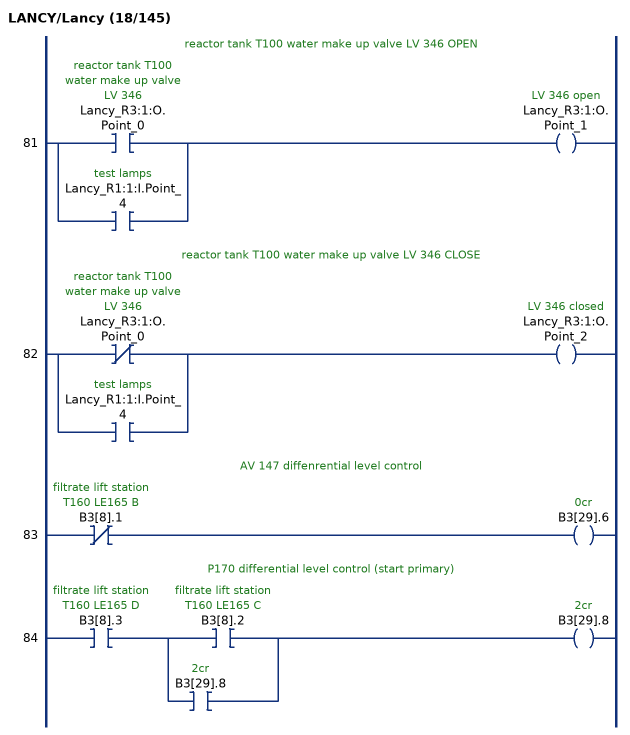
   // reactor tank T100 water make up valve LV 346 OPEN
   81: [XIC(Lancy_R3:1:O.Point_0) ,XIC(Lancy_R1:1:I.Point_4) ]OTE(Lancy_R3:1:O.Point_1);
   // reactor tank T100 water make up valve LV 346 CLOSE
   82: [XIO(Lancy_R3:1:O.Point_0) ,XIC(Lancy_R1:1:I.Point_4) ]OTE(Lancy_R3:1:O.Point_2);
   // AV 147 diffenrential level control
   83: XIO(B3[8].1)OTE(B3[29].6);
   // P170 differential level control (start primary)
   84: XIC(B3[8].3)[XIC(B3[8].2) ,XIC(B3[29].8) ]OTE(B3[29].8);
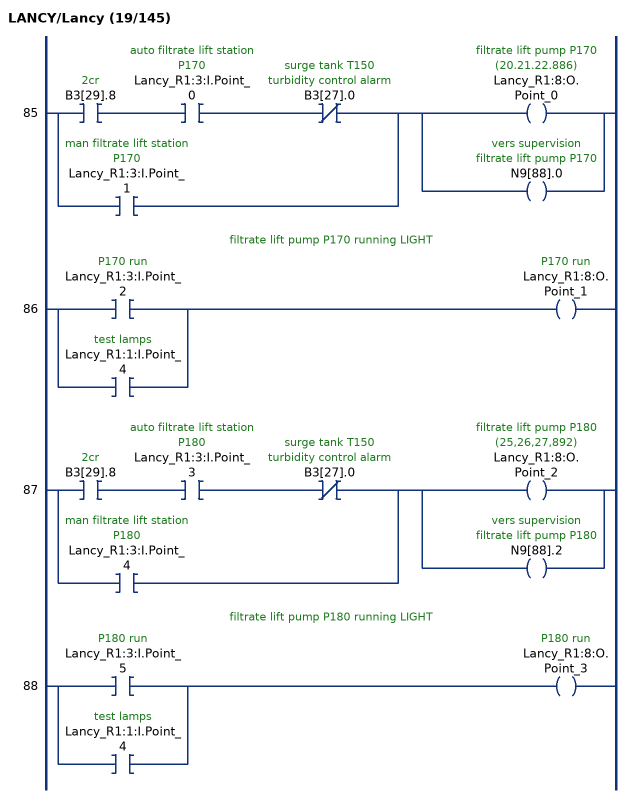
   85: [XIC(B3[29].8) XIC(Lancy_R1:3:I.Point_0) XIO(B3[27].0) ,XIC(Lancy_R1:3:I.Point_1) ][OTE(Lancy_R1:8:O.Point_0) ,OTE(N9[88].0) ];
   // filtrate lift pump P170 running LIGHT
   86: [XIC(Lancy_R1:3:I.Point_2) ,XIC(Lancy_R1:1:I.Point_4) ]OTE(Lancy_R1:8:O.Point_1);
   87: [XIC(B3[29].8) XIC(Lancy_R1:3:I.Point_3) XIO(B3[27].0) ,XIC(Lancy_R1:3:I.Point_4) ][OTE(Lancy_R1:8:O.Point_2) ,OTE(N9[88].2) ];
   // filtrate lift pump P180 running LIGHT
   88: [XIC(Lancy_R1:3:I.Point_5) ,XIC(Lancy_R1:1:I.Point_4) ]OTE(Lancy_R1:8:O.Point_3);
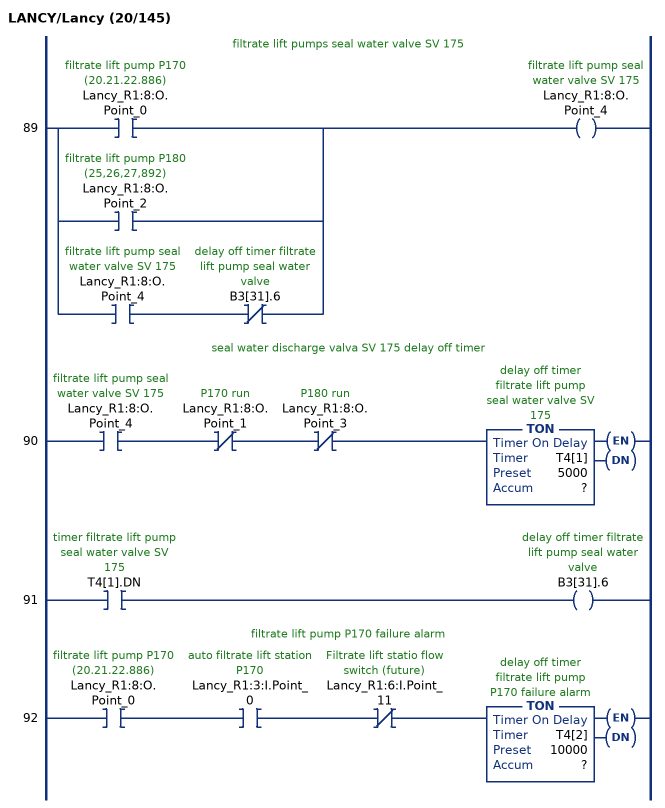
   // filtrate lift pumps seal water valve SV 175
   89: [[XIC(Lancy_R1:8:O.Point_0) ,XIC(Lancy_R1:8:O.Point_2) ] ,XIC(Lancy_R1:8:O.Point_4) XIO(B3[31].6) ]OTE(Lancy_R1:8:O.Point_4);
   // seal water discharge valva SV 175 delay off timer
   90: XIC(Lancy_R1:8:O.Point_4)XIO(Lancy_R1:8:O.Point_1)XIO(Lancy_R1:8:O.Point_3)TON(T4[1],?,?);
   91: XIC(T4[1].DN)OTE(B3[31].6);
   // filtrate lift pump P170 failure alarm
   92: XIC(Lancy_R1:8:O.Point_0)XIC(Lancy_R1:3:I.Point_0)XIO(Lancy_R1:6:I.Point_11)TON(T4[2],?,?);
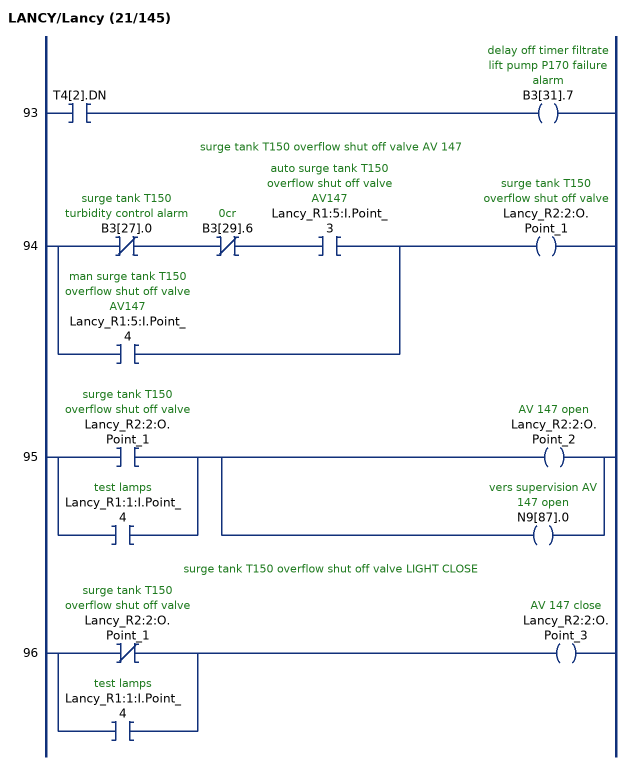
   93: XIC(T4[2].DN)OTE(B3[31].7);
   // surge tank T150 overflow shut off valve AV 147
   94: [XIO(B3[27].0) XIO(B3[29].6) XIC(Lancy_R1:5:I.Point_3) ,XIC(Lancy_R1:5:I.Point_4) ]OTE(Lancy_R2:2:O.Point_1);
   95: [XIC(Lancy_R2:2:O.Point_1) ,XIC(Lancy_R1:1:I.Point_4) ][OTE(Lancy_R2:2:O.Point_2) ,OTE(N9[87].0) ];
   // surge tank T150 overflow shut off valve LIGHT CLOSE
   96: [XIO(Lancy_R2:2:O.Point_1) ,XIC(Lancy_R1:1:I.Point_4) ]OTE(Lancy_R2:2:O.Point_3);
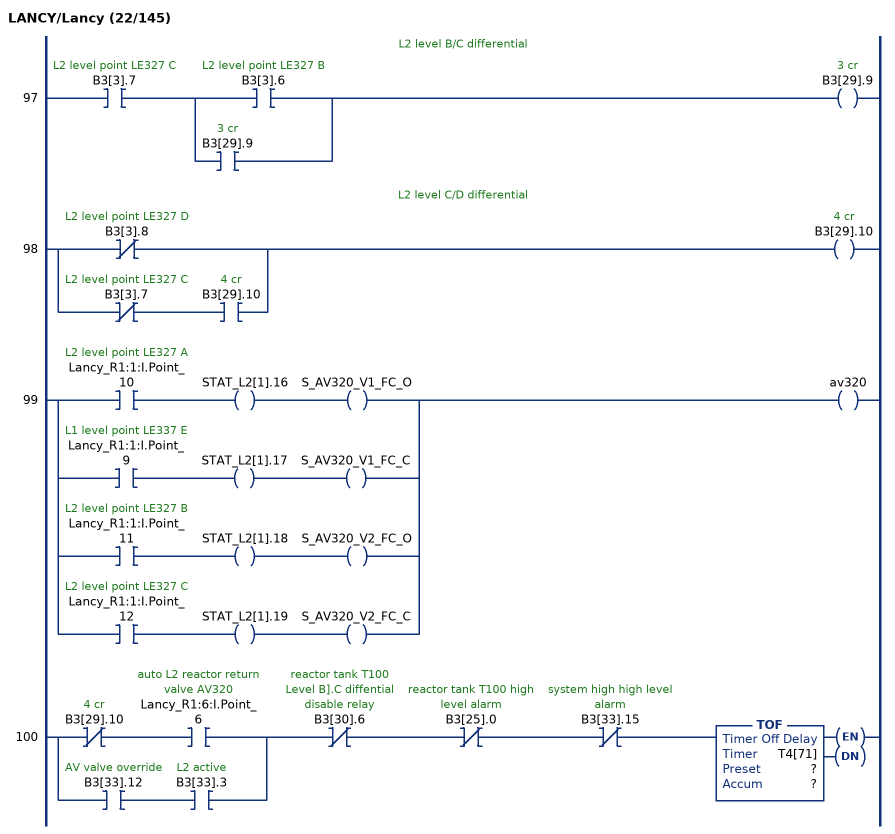
   // L2 level B/C differential
   97: XIC(B3[3].7)[XIC(B3[3].6) ,XIC(B3[29].9) ]OTE(B3[29].9);
   // L2 level C/D differential
   98: [XIO(B3[3].8) ,XIO(B3[3].7) XIC(B3[29].10) ]OTE(B3[29].10);
   99: [XIC(Lancy_R1:1:I.Point_10) OTE(STAT_L2[1].16) OTE(S_AV320_V1_FC_O) ,XIC(Lancy_R1:1:I.Point_9) OTE(STAT_L2[1].17) OTE(S_AV320_V1_FC_C) ,XIC(Lancy_R1:1:I.Point_11) OTE(STAT_L2[1].18) OTE(S_AV320_V2_FC_O) ,XIC(Lancy_R1:1:I.Point_12) OTE(STAT_L2[1].19) OTE(S_AV320_V2_FC_C) ]OTE(av320);
   100: [XIO(B3[29].10) XIC(Lancy_R1:6:I.Point_6) ,XIC(B3[33].12) XIC(B3[33].3) ]XIO(B3[30].6)XIO(B3[25].0)XIO(B3[33].15)TOF(T4[71],?,?);
